// TwinCAT 3 PLC project Untitled1
// ProgramVersion: 3.1.4023.0
// libraries:
//   Tc2_Standard, * (Beckhoff Automation GmbH)
//   Tc2_System, * (Beckhoff Automation GmbH)
//   Tc2_Utilities, * (Beckhoff Automation GmbH)
//   Tc3_Database, * (Beckhoff Automation GmbH)
//   Tc3_EventLogger, * (Beckhoff Automation GmbH)
//   Tc3_Module, * (Beckhoff Automation GmbH)
// project tree:
//   DUTs/DataFlowManagement/ ST_NovRam.TcDUT
//   DUTs/DataFlowManagement/ST_NovRam_SubST/ E_DB_StructureType.TcDUT, ST_NovRam_Status.TcDUT, ST_FileRingBuffer_Status.TcDUT
//   DUTs/ErrHandle/ E_DataBaseTable.TcTLEO
//   DUTs/ E_DataBaseStatus.TcDUT, E_DBID.TcDUT, E_DB_DataType.TcDUT, E_RegularCheckSensorResult.TcDUT, ST_AlarmInfo_DB.TcDUT, ST_AlarmInfo_DB_save.TcDUT, ST_HardwareConfigure_DB.TcDUT, ST_MachineInformation.TcDUT, ST_MachineParameter.TcDUT, ST_MessageElement.TcDUT, ST_OEE_ProductionReport.TcDUT, ST_OEE_ProductionSummary.TcDUT, ST_RegularCheck_Results.TcDUT, ST_RegularCheck_Results_DB.TcDUT, ST_ShopOrderInformation.TcDUT, ST_SoDuration.TcDUT, ST_StopCount.TcDUT
//   DUTs/PHI/ ST_CmdPara_PHI_DB.TcDUT, ST_Inspection_DB.TcDUT, ST_PHI_GroupData_DB.TcDUT, ST_Production_History_DB.TcDUT, ST_Production_History_DB_Test.TcDUT
//   GVLs/ GVL.TcGVL
//   / PlcTask.TcTTO, Task_Consumer.TcTTO
//   POUs/ CheckBounds.TcPOU, MAIN.TcPOU, PG_AddData.TcPOU, PG_SaveData.TcPOU
//   POUs/DataFlow/Lv1/ FB_DataFlowManagement.TcPOU
//   POUs/DataFlow/Lv2/ FB_DataToNovRam.TcPOU, FB_FileRingBufferToDB.TcPOU, FB_NovRamToFileRingBuffer.TcPOU
//   POUs/DataFlow/Lv3%28DB%29/Lv1/ FB_DataUpload_Leo.TcPOU (not stored)
//   POUs/DataFlow/Lv3%28DB%29/Lv2/Background/ FB_CheckDBconnection_DB.TcPOU (not stored)
//   POUs/DataFlow/Lv3%28DB%29/Lv2/DB/ FB_AlarmHistory_DB.TcPOU (not stored), FB_OEE_ProductionReport_DB.TcPOU (not stored), FB_OEE_ProductionSummary_DB.TcPOU (not stored), FB_ProductionHistoryInspection_DB.TcPOU (not stored), FB_Regular_Check_Results_DB.TcPOU (not stored), FB_SoDuration_DB.TcPOU (not stored), FB_StopCount_DB.TcPOU (not stored)
// real-time tasks:
//   TASK PlcTask: cycle T#1ms, priority 20, ADS port 350
//   TASK Task 4: cycle T#1ms, priority 1, ADS port 351

CONFIGURATION Untitled1
    RESOURCE PLC ON TwinCAT3
        TASK PlcTask(INTERVAL := T#1ms, PRIORITY := 20);
        TASK Task_Consumer(INTERVAL := T#1ms, PRIORITY := 1);
        PROGRAM MAIN WITH PlcTask : MAIN;
        PROGRAM PG_AddData WITH PlcTask : PG_AddData;
        PROGRAM PG_SaveData WITH Task_Consumer : PG_SaveData;
    END_RESOURCE
END_CONFIGURATION

// ---- DUTs/DataFlowManagement/ST_NovRam.TcDUT
TYPE ST_NovRam :
STRUCT
	
	//Status
	//NovRam_Status:ST_NovRam_Status;
	arrNovRam_Status:ARRAY[0..6] OF ST_NovRam_Status;
	//FileRingBuffer_Status:ST_FileRingBuffer_Status;
	arrFileRingBuffer_Status:ARRAY[0..6] OF ST_FileRingBuffer_Status;
	
	
	
	//Compressed DATA
	AlarmHistory:ARRAY [0..GVL.NovRamBufferRatio-1] OF ARRAY [0..GVL.arrArrayLength[E_DB_StructureType.AlarmHistory]-1] OF ST_AlarmInfo_DB_save;
	ProductionHistory:ARRAY [0..GVL.NovRamBufferRatio-1] OF ARRAY [0..GVL.arrArrayLength[E_DB_StructureType.ProductionHistory]-1] OF ST_PHI_GroupData_DB;
	ProductionReport:ARRAY [0..GVL.NovRamBufferRatio-1]OF ARRAY [0..GVL.arrArrayLength[E_DB_StructureType.ProductionReport]-1] OF ST_OEE_ProductionReport;
	ProductionSummary:ARRAY [0..GVL.NovRamBufferRatio-1]OF ARRAY [0..GVL.arrArrayLength[E_DB_StructureType.ProductionSummary]-1] OF ST_OEE_ProductionSummary;
	SoDuration:ARRAY [0..GVL.NovRamBufferRatio-1]OF ARRAY [0..GVL.arrArrayLength[E_DB_StructureType.SoDuration]-1] OF ST_SoDuration;
	StopCount:ARRAY [0..GVL.NovRamBufferRatio-1]OF ARRAY [0..GVL.arrArrayLength[E_DB_StructureType.StopCount]-1] OF ST_StopCount;
	RegularCheckResults:ARRAY [0..GVL.NovRamBufferRatio-1]OF ARRAY [0..GVL.arrArrayLength[E_DB_StructureType.RegularCheckResults]-1] OF ST_RegularCheck_Results;
	

END_STRUCT
END_TYPE

// ---- DUTs/DataFlowManagement/ST_NovRam_SubST/E_DB_StructureType.TcDUT
{attribute 'qualified_only'}
{attribute 'strict'}
TYPE E_DB_StructureType :
(
	AlarmHistory := 0,
	ProductionHistory := 1,
	ProductionReport := 2,
	ProductionSummary := 3,
	SoDuration:=4,
	StopCount:=5,
	RegularCheckResults:=6
);
END_TYPE

// ---- DUTs/DataFlowManagement/ST_NovRam_SubST/ST_NovRam_Status.TcDUT
TYPE ST_NovRam_Status :
STRUCT
	nowRowIndex:UDINT;
	writenIndex:UDINT;
	RowDataLocked:ARRAY[0..GVL.NovRamBufferRatio-1]OF BOOL;
	writenCount:UDINT;//1217
	
END_STRUCT
END_TYPE

// ---- DUTs/DataFlowManagement/ST_NovRam_SubST/ST_FileRingBuffer_Status.TcDUT
TYPE ST_FileRingBuffer_Status :
STRUCT
	bFileFull:ARRAY[0..GVL.NovRamBufferRatio-1] OF ARRAY [0..GVL.FileRingBufferRatio-1] OF BOOL;//9
	
	//FileRingBufferLocked:ARRAY[0..GVL.FileRingBufferTotalNum-1]OF BOOL;
	nowFileIndex:ARRAY [0..gvl.FileRingBufferRatio-1] OF UDINT;//3
END_STRUCT
END_TYPE

// ---- DUTs/ErrHandle/E_DataBaseTable.TcTLEO
{attribute 'qualified_only'}
{attribute 'to_string'}
TYPE E_DataBaseTable :
(
	NoError := 0,
	HardwareConfig_ReadFail,
	HardwareConfig_ReadDataOutOfRange,
	HardwareConfig_InputReferenceInvaild,
	HardwareConfig_NoData,
	MachineParameter_ReadFail,
	MachineParameter_ReadDataOutOfRange,
	MachineParameter_InputReferenceInvaild,
	MachineParameter_NoData,
	MachineParameter_FillDataToSubsysFail,
	MachineParameter_FillDataToCoreSysFail,
	MachineParameter_FillDataToMachineFail,
	MessageList_ReadFail,
	MessageList_ReadDataOutOfRange,	
	MessageList_InputReferenceInvaild,
	MessageList_NoData,
	MessageList_MessageCodeOrArraySizeOutOfRange,
	AlarmHistory_UploadDataFail,
	DataUpload_ConnectToDBFail,
	DataUpload_AlarmHistoryBufferFull,
	DataUpload_AlarmHistoryUploadFail,
	DataUpload_AlarmHistoryUploadFailWriteDataToFileFail, //重大異常，不能直接reset需要人員排查原因，程式內部鎖死不能reset
	DataUpload_ProductionHistoryBufferFull,
	DataUpload_ProductionHistoryUploadFail,
	DataUpload_ProductionHistoryWriteDataToFileFail, //重大異常，不能直接reset需要人員排查原因，程式內部鎖死不能reset
	DataUpload_ProductionReportBufferFull,
	DataUpload_ProductionReportUploadFail,
	DataUpload_ProductionReportWriteDataToFileFail, //重大異常，不能直接reset需要人員排查原因，程式內部鎖死不能reset
	DataUpload_ProductionSummaryBufferFull,
	DataUpload_ProductionSummaryUploadFail,
	DataUpload_ProductionSummaryWriteDataToFileFail, //重大異常，不能直接reset需要人員排查原因，程式內部鎖死不能reset
	DataUpload_SoDurationBufferFull,
	DataUpload_SoDurationUploadFail,
	DataUpload_SoDurationWriteDataToFileFail, //重大異常，不能直接reset需要人員排查原因，程式內部鎖死不能reset
	DataUpload_StopCountBufferFull,	
	DataUpload_StopCountUploadFail,
	DataUpload_StopCountWriteDataToFileFail, //重大異常，不能直接reset需要人員排查原因，程式內部鎖死不能reset
	DataUpload_RegularCheckResultsBufferFull,
	DataUpload_RegularCheckResultsUploadFail,
	DataUpload_RegularCheckResultsWriteDataToFileFail, //重大異常，不能直接reset需要人員排查原因，程式內部鎖死不能reset
	ProductionReport_UploadDataFail,
	ProductionSummary_UploadDataFail,
	ProductionHistoryInspection_UploadDataFail,
	RegularCheckResults_UploadDataFail,
	SoDuration_UploadDataFail,
	StopCount_UploadDataFail,
	CheckDBconnection_ReadDBStatusTimeout,
	CheckDBconnection_RetryConnectToDBFail,
	CheckDBconnection_StatusDataOutOfRange,
	ProdHistoryProcedure_UploadDataFail,
	ProdHistoryProcedure_WriteDataToFileFail, //重大異常，不能直接reset需要人員排查原因，程式內部鎖死不能reset
	ProdHistoryProcedure_InputInterfaceInvalid,
	ProdStatusChangedStopCount_FillDataTimeout,
	ProdStatusChangedStopCount_AddDataToBufferTimeout,
	UploadEndBatchData_FillProductionReportDataTimeout,
	UploadEndBatchData_FillProductionSummaryDataTimeout,
	UploadEndBatchData_FillSoDurationDataTimeout,
	UploadEndBatchData_AddProductionReportDataToBufferTimeout,
	UploadEndBatchData_AddProductionSummaryDataToBufferTimeout,
	UploadEndBatchData_AddSoDurationDataToBufferTimeout,
	UploadProdRegularReport_FillProductionReportDataTimeout,
	UploadProdRegularReport_AddProductionReportDataToBufferTimeout
	
	
)UDINT;
END_TYPE

// ---- DUTs/E_DataBaseStatus.TcDUT
{attribute 'qualified_only'}
{attribute 'to_string'}
TYPE E_DataBaseStatus :
(
	ONLINE := 0,
	RESTORING,
	RECOVERING,
	RECOVERY_PENDING,
	SUSPECT,
	EMERGENCY,
	OFFLINE,
	COPYING,
	OFFLINE_SECONDARY
)USINT;
END_TYPE

// ---- DUTs/E_DBID.TcDUT
{attribute 'qualified_only'}
{attribute 'to_string'}
TYPE E_DBID :
(
	BypassDB	:= 0,
	RemoteDB  	:= 1,
	LocalDB		:= 2
)UDINT;
END_TYPE

// ---- DUTs/E_DB_DataType.TcDUT
{attribute 'qualified_only'}
{attribute 'to_string'}
TYPE E_DB_DataType :
(
	Double := 0,
	StringType,
	Ring,
	Boolean,
	I32,
	U32,
	DynamicRing
)INT;
END_TYPE

// ---- DUTs/E_RegularCheckSensorResult.TcDUT
{attribute 'qualified_only'}
{attribute 'to_string'}
TYPE E_RegularCheckSensorResult :
(
	Null, // 感測器沒判定過/使用  DB寫Null
	Pass, // 判定結果為OK  DB寫1
	Fail // 判定結果為NG  DB寫0
);
END_TYPE

// ---- DUTs/PHI/ST_CmdPara_PHI_DB.TcDUT
TYPE ST_CmdPara_PHI_DB :
	STRUCT
		//Product History
		dt_start_time            : DT ;
		r_duration               : REAL ;
		dt_end_time              : DT ;
		di_station_number        : DINT ;
		wstr_station_name        : WSTRING(255) ; //20221107
		di_track_number          : DINT ;
		di_wpc_number            : DINT ;
		b_part_ok_overal_results : BOOL ;
		str_so_number            : STRING(12) ;
		str_faam_id              : STRING(20) ;
		di_so_id                 : DINT ;
		
		//1st Inspection
		di_sub_station_number_1 : DINT ;
		str_sensor_type_1       : STRING(50) ;
		b_inspection_results_1  : BOOL ;
		r_inspection_value_1    : REAL ;
		str_faam_id_1           : STRING(20) ;
		str_so_number_1         : STRING(12) ;
		
		//2nd Inspection
		di_sub_station_number_2 : DINT ;
		str_sensor_type_2       : STRING(50) ;
		b_inspection_results_2  : BOOL ;
		r_inspection_value_2    : REAL ;
		str_faam_id_2           : STRING(20) ;
		str_so_number_2         : STRING(12) ;
		
		//3nd Inspection
		di_sub_station_number_3 : DINT ;
		str_sensor_type_3       : STRING(50) ;
		b_inspection_results_3  : BOOL ;
		r_inspection_value_3    : REAL ;
		str_faam_id_3           : STRING(20) ;
		str_so_number_3         : STRING(12) ;
		
		//4nd Inspection
		di_sub_station_number_4 : DINT ;
		str_sensor_type_4	     : STRING(50) ;
		b_inspection_results_4  : BOOL ;
		r_inspection_value_4    : REAL ;
		str_faam_id_4           : STRING(20) ;
		str_so_number_4         : STRING(12) ;
		
		//5nd Inspection
		di_sub_station_number_5 : DINT ;
		str_sensor_type_5       : STRING(50) ;
		b_inspection_results_5  : BOOL ;
		r_inspection_value_5    : REAL ;
		str_faam_id_5           : STRING(20) ;
		str_so_number_5         : STRING(12) ;
	END_STRUCT
END_TYPE

// ---- DUTs/PHI/ST_Inspection_DB.TcDUT
TYPE ST_Inspection_DB : // Sensor inspection information and result
	STRUCT
		diSub_station_number 	: DINT ;			// 站點上第N組感測器
		sSensor_type        	: STRING(50) ;	// Sensor類型
		bInspection_results 	: BOOL ;			// Sensor回傳結果
		rInspection_value   	: REAL ;			// Sensor回傳數值
		sFaam_id            	: STRING(20) ;
		sSo_number          	: STRING(12) ;
		//product_history_id 	: LINT ;
	END_STRUCT
END_TYPE

// ---- DUTs/PHI/ST_PHI_GroupData_DB.TcDUT
 //Product History and Inspection data
 //X64 size: 1064 bytes
TYPE ST_PHI_GroupData_DB : //Production information of the station, including single production data and sensor results
	STRUCT
		stProductHistory        						: ST_Production_History_DB ; // single production data
		arrstInspection         						: ARRAY[1..5] OF ST_Inspection_DB ; //max sensor number = 5
		arrbInspectionResultHaveSensorValue           	: ARRAY[1..5] OF BOOL ; // return data of the sensor have a numerical value
	END_STRUCT
END_TYPE

// ---- DUTs/PHI/ST_Production_History_DB.TcDUT
TYPE ST_Production_History_DB : // single production data of a station
	STRUCT
		dtStart_time             	: DT ;					// 作業開始時間
		rDuration               	: REAL ;				// unit: sec    (end_time - start_time)
		dtEnd_time               	: DT ;					// 作業結束時間
		diStation_number         	: DINT ;				// 站點編號
		wsStation_name           	: WSTRING(255) ; 		// 站點名稱
		diTrack_number           	: DINT ;				// 未定義  Smart Hardcode為1
		diWpc_number            	: DINT ;				// Shuttle Id
		bPart_ok_overal_results 	: BOOL ;				// 此站點最終判斷/作業結果為OK或NG (彙整站點上的感測器結果及作業結果)
		sSo_number              	: STRING(12) ;			// 由HMI透過ADS告知  (DB中的So資料表需要存在對應資料)
		sFaam_id                	: STRING(20) ;			// 由DB讀取
		diSo_id                  	: DINT ;				// 由HMI透過ADS告知 (DB中的So資料表需要存在對應資料)
	END_STRUCT
END_TYPE

// ---- DUTs/PHI/ST_Production_History_DB_Test.TcDUT
TYPE ST_Production_History_DB_Test: // single production data of a station
	STRUCT
		dtStart_time             	: DT ;					// 作業開始時間
		rDuration               	: REAL ;				// unit: sec    (end_time - start_time)
		dtEnd_time               	: DT ;					// 作業結束時間
		usiStation_number         	: USINT ;				// 站點編號
		sStation_name           	: STRING(50) ; 		// 站點名稱
		usiTrack_number           	: USINT ;				// 未定義  Smart Hardcode為1
		usiWpc_number            	: USINT ;				// Shuttle Id
		bPart_ok_overal_results 	: BOOL ;				// 此站點最終判斷/作業結果為OK或NG (彙整站點上的感測器結果及作業結果)
		sSo_number              	: STRING(12) ;			// 由HMI透過ADS告知  (DB中的So資料表需要存在對應資料)
		sFaam_id                	: STRING(20) ;			// 由DB讀取
		diSo_id                  	: DINT ;				// 由HMI透過ADS告知 (DB中的So資料表需要存在對應資料)
	END_STRUCT
END_TYPE

// ---- DUTs/ST_AlarmInfo_DB.TcDUT
// X64 size: 4984 byte
TYPE ST_AlarmInfo_DB :
STRUCT
	lrTime_ms    	: LREAL ;		
	iMsgProc    	: INT ;			// 未明 先填1
	iStateAfter 	: INT ;			// 1: Error trigger  0: reset
	iMsgClass   	: INT ;			// 1: error 2: warning 3: msg
	diMsgNumber  	: DINT ;		// MsgCode等同於ErrorId
	wsVar1			: WSTRING(255);	// 備註1(可不填)
	wsVar2			: WSTRING(255);	// 備註2(可不填)
	wsVar3			: WSTRING(255);	// 備註3(可不填)
	wsVar4			: WSTRING(255);	// 備註4(可不填)
	wsVar5			: WSTRING(255);	// 備註5(可不填)
	wsVar6			: WSTRING(255);	// 備註6(可不填)
	wsVar7			: WSTRING(255);	// 備註7(可不填)
	wsVar8			: WSTRING(255);	// 備註8(可不填)
	sTimeString 	: STRING(25); 	// Data Format: '2023-08-15 15:11:14'  		// SQL Database為char type 26bytes 
	wsMsgText    	: WSTRING(255); // 文字訊息(顯示在HMI給使用者看的訊息)
	sPLC        	: STRING(255); 	// Data Format: 'CoreSys' 
	wsEquipment  	: WSTRING(25);
	sFaam_id    	: STRING(20);
	
END_STRUCT
END_TYPE

// ---- DUTs/ST_AlarmInfo_DB_save.TcDUT
// X64 size: 680 byte
TYPE ST_AlarmInfo_DB_save:
STRUCT
	(*
	lrTime_ms    	: LREAL ;		
	siMsgProc    	: SINT ;			// 未明 先填1
	siStateAfter 	: SINT ;			// 1: Error trigger  0: reset
	siMsgClass   	: SINT ;			// 1: error 2: warning 3: msg
	diMsgNumber  	: DINT ;		// MsgCode等同於ErrorId
	//wsVar1			: WSTRING(255);	// 備註1(可不填)
	//wsVar2			: WSTRING(255);	// 備註2(可不填)
	//wsVar3			: WSTRING(255);	// 備註3(可不填)
	//wsVar4			: WSTRING(255);	// 備註4(可不填)
	//wsVar5			: WSTRING(255);	// 備註5(可不填)
	//wsVar6			: WSTRING(255);	// 備註6(可不填)
	//wsVar7			: WSTRING(255);	// 備註7(可不填)
	//wsVar8			: WSTRING(255);	// 備註8(可不填)
	sTimeString 	: STRING(25); 	// Data Format: '2023-08-15 15:11:14'  		// SQL Database為char type 26bytes 
	wsMsgText    	: WSTRING(255); // 文字訊息(顯示在HMI給使用者看的訊息)
	sPLC        	: STRING(50); 	// Data Format: 'CoreSys' 
	wsEquipment  	: WSTRING(25);
	sFaam_id    	: STRING(20);
	*)
	lrTime_ms    	: LREAL ;		
	iMsgProc    	: INT ;			// 未明 先填1
	iStateAfter 	: INT ;			// 1: Error trigger  0: reset
	iMsgClass   	: INT ;			// 1: error 2: warning 3: msg
	diMsgNumber  	: DINT ;		// MsgCode等同於ErrorId
	sTimeString 	: STRING(25); 	// Data Format: '2023-08-15 15:11:14'  		// SQL Database為char type 26bytes 
	wsMsgText    	: WSTRING(255); // 文字訊息(顯示在HMI給使用者看的訊息)
	sPLC        	: STRING(255); 	// Data Format: 'CoreSys' 
	wsEquipment  	: WSTRING(25);
	sFaam_id    	: STRING(20);
END_STRUCT
END_TYPE

// ---- DUTs/ST_HardwareConfigure_DB.TcDUT
TYPE ST_HardwareConfigure_DB :
STRUCT
	iParametersID			: INT;
	wsConfigureItem			: WSTRING(255);
	wsConfigureName			: WSTRING(255);
	wsConfigureValue		: WSTRING(255);
	wsDataType				: WSTRING(255);
	wsDescription			: WSTRING(255);
END_STRUCT
END_TYPE

// ---- DUTs/ST_MachineInformation.TcDUT
TYPE ST_MachineInformation :
STRUCT
	sFaam_id                  : STRING(20) ;	// 設備ID
	wsEquipment               : WSTRING(25) ;	// 設備名稱
END_STRUCT
END_TYPE

// ---- DUTs/ST_MachineParameter.TcDUT
// Generated by SQL Query Editor
TYPE ST_MachineParameter :
STRUCT
	iParameters_Index	: INT;
	wsTag_Name			: WSTRING(255);
	iStation			: INT;
	wsParameters_Unit	: WSTRING(50);
	iPackTagID			: INT;
	wsParameters_Value	: WSTRING(255);
	eDataType			: E_DB_DataType;
END_STRUCT
END_TYPE


//SQL Command
(*
SELECT          Global_Machine_Parameters.Parameters_Index, 
				Global_Machine_Parameters.Parameters_Name, 
				Global_Machine_Parameters.Station, 
				Global_Machine_Parameters.Parameters_Unit,
                Global_Machine_Parameters.PackTagID, 
				Global_Machine_Parameters_Value.Parameters_Value
FROM            Global_Machine_Parameters_Value INNER JOIN
                Global_Machine_Parameters ON 
                Global_Machine_Parameters_Value.Parameters_Index = Global_Machine_Parameters.Parameters_Index
ORDER BY Global_Machine_Parameters.Parameters_Index
*)

// ---- DUTs/ST_MessageElement.TcDUT
// X64 Size: 2052 byte
TYPE ST_MessageElement :
STRUCT
	iCode						: INT;			// MsgCode (ErrorCode)
	wsCategory					: WSTRING(255); // 文字訊息分類 EX: "Safety Message", "Beaker and Bin and Drawer Message" etc.
	wsItem						: WSTRING(255);	// 此訊息的項目名稱，通常會與wsFirst_Language_Message重複
	wsFirst_Language_Message  	: WSTRING(255); // 多國語言1文字訊息(此項為預設值 內文為英文)
	wsSecond_Language_Message 	: WSTRING(255); // 多國語言2文字訊息(內文為中文或其他)
	iMessage_Type 				: INT;
END_STRUCT
END_TYPE

// ---- DUTs/ST_OEE_ProductionReport.TcDUT
// X64 size: 172 bytes
TYPE ST_OEE_ProductionReport :
	STRUCT
		wsOee_equipment            	: WSTRING(25) ;
		dtTime_start               	: DT ;
		dtTime_end                 	: DT ;
		diAverage_ppm              	: DINT ;
		diIdeal_production         	: DINT ;
		diOk_part_count            	: DINT ;
		rTotal_idle_time          	: REAL ;
		diReal_production          	: DINT ;
		diGood_parts               	: DINT ;
		rGood_parts_percentage    	: REAL ;
		diQuantity_loss            	: DINT ;
		rQuantity_loss_percentage 	: REAL ;
		rPm                       	: REAL ;
		rYm                       	: REAL ;
		rAm                       	: REAL ;
		rEm                       	: REAL ;
		rOm                       	: REAL ;
		rAvailable_time           	: REAL ;
		rSchedule_loss            	: REAL ;
		rRunning_time             	: REAL ;
		rDowntime_loss            	: REAL ;
		sFaam_id                  	: STRING(20) ;
		sSo_number               	: STRING(12) ;
		diSo_id                    	: DINT ;
	END_STRUCT
END_TYPE

// ---- DUTs/ST_OEE_ProductionSummary.TcDUT
// X64 size: 148 bytes
TYPE ST_OEE_ProductionSummary :
	STRUCT
		wsEquipment     : WSTRING(20) ;
		wsSummary_type  : WSTRING(30) ;
		diSummary_value : DINT ;
		sFaam_id       : STRING(20) ;
		sSo_number     : STRING(12) ;
		diSo_id         : DINT ;
	END_STRUCT
END_TYPE

// ---- DUTs/ST_RegularCheck_Results.TcDUT
// X64 size: 572 bytes
TYPE ST_RegularCheck_Results :
	STRUCT
		diStation_number          	: DINT ;
		diTrack_number            	: DINT ;
		dtStart_time              	: DT ;
		eSensor                  	: E_RegularCheckSensorResult ;
		eCamera                  	: E_RegularCheckSensorResult ;
		eLoadcell                	: E_RegularCheckSensorResult ;
		eSensor2                 	: E_RegularCheckSensorResult ;
		diRegular_check_id        	: DINT ;
		sFaam_id                 	: STRING(20) ;
		sSo_number               	: STRING(12) ;
		diSo_id                   	: DINT ;
		wsEmployee_name_logged_in 	: WSTRING(255) ;
	END_STRUCT
END_TYPE

// ---- DUTs/ST_RegularCheck_Results_DB.TcDUT
// X64 size: 572 bytes
TYPE ST_RegularCheck_Results_DB :
	STRUCT
		diStation_number          	: DINT ;
		diTrack_number            	: DINT ;
		dtStart_time              	: DT ;
		bSensor                  	: BOOL ;
		bCamera                  	: BOOL ;
		bLoadcell                	: BOOL ;
		bSensor2                 	: BOOL ;
		diRegular_check_id        	: DINT ;
		sFaam_id                 	: STRING(20) ;
		sSo_number               	: STRING(12) ;
		diSo_id                   	: DINT ;
		wsEmployee_name_logged_in 	: WSTRING(255) ;
	END_STRUCT
END_TYPE

// ---- DUTs/ST_ShopOrderInformation.TcDUT
TYPE ST_ShopOrderInformation :
STRUCT
	diSo_id                    	: DINT ;
	sSo_number               	: STRING(12) ;
END_STRUCT
END_TYPE

// ---- DUTs/ST_SoDuration.TcDUT
// X64 size: 2100 bytes
TYPE ST_SoDuration :
	STRUCT
		dtBatch_start_time            	: DT ;
		dtBatch_end_time              	: DT ;
		//bNormal_complition           	: BOOL ; //改放至最後才寫  放在這位置寫入DB時會導致下個資料WString在DB裡開頭多一個空白byte的資料
		wsBatch_end_reason             	: WSTRING(255) ;
		wsBatch_end_reason_description 	: WSTRING(255) ;
		wsEmployee_name_start_user     	: WSTRING(255) ;
		wsEmployee_name_end_user       	: WSTRING(255) ;
		sSo_number                    	: STRING(12) ;
		sFaam_id                      	: STRING(20) ;
		diSo_id                        	: DINT ;
		bNormal_complition           	: BOOL ;
	END_STRUCT
END_TYPE

// ---- DUTs/ST_StopCount.TcDUT
TYPE ST_StopCount :
	STRUCT
		dtStart_time              : DT ;
		dtEnd_time                : DT ;
		wsEmployee_name_logged_in : WSTRING(255) ;
		sStop_reason             : STRING(3) ;
		sAssembly_income_code    : STRING(16) ;
		sSo_number               : STRING(12) ;
		sFaam_id                 : STRING(20) ;
		diSo_id                   : DINT ;
		wsEquipment               : WSTRING(25) ;
	END_STRUCT
END_TYPE

// ---- GVLs/GVL.TcGVL
{attribute 'qualified_only'}
VAR_GLOBAL CONSTANT//NovRam Management
		
	Max_IndexNum:UDINT:=40;//Index數量

	//File大小
	//fileRingBufferSize:UDINT:=50*1000;//Byte
	arrFileRingBufferSize:ARRAY [0..6] OF UDINT:=[
	100*1000,//Alarm History
	100*1000,//Production History
	100*1000,//ProductionReport
	100*1000,//ProductionSummary
	100*1000,//SoDuration
	100*1000,//StopCount
	100*1000//RegularCheckResults
	];
	
	//資料的陣列長度
	//AlarmHistory_ArrayLength:UDINT:=30;
	//ProductionHistory_ArrayLength:UDINT:=30;
	arrArrayLength:ARRAY[0..6] OF UDINT:=[
	30,//Alarm History
	30,//Production History
	30,//ProductionReport
	30,//ProductionSummary
	30,//SoDuration
	30,//StopCount
	30//RegularCheckResults
	];
	
	//NovRam中Array數量
	NovRamBufferRatio:UDINT:=3;
	//arrNovRamBufferRatio:ARRAY [0..1] OF UDINT:=[
	//3,//Alarm History
	//3//Production History
	//];
	
	//單一NovRam Array對應的File數量
	FileRingBufferRatio:UDINT:=3;
	//arrFileRingBufferRatio:ARRAY[0..1] OF UDINT:=[
	//10,//Alarm History
	//10//Production History
	//];
	
	//fileFolder:STRING(255):='c:\_Yenlin\';
	arrFileFolder:ARRAY [0..6] OF STRING(255):=[
	'c:\_Yenlin\',//Alarm History
	'c:\_Yenlin\',//Production History
	'c:\_Yenlin\',//ProductionReport
	'c:\_Yenlin\',//ProductionSummary
	'c:\_Yenlin\',//SoDuration
	'c:\_Yenlin\',//StopCount
	'c:\_Yenlin\'//RegularCheckResults
	];
	
	
END_VAR

VAR_GLOBAL
	fbDataFlowManagement:FB_DataFlowManagement;
	udiUpperCnt : UDINT;
	udiLowerCnt	: UDINT;
END_VAR

// ---- POUs/MAIN.TcPOU
PROGRAM MAIN
VAR
	i:UDINT;
	
END_VAR

END_PROGRAM

// ---- POUs/PG_AddData.TcPOU
PROGRAM PG_AddData
VAR
	i:UDINT;
	repeatTimer:TON;
	
	
	AlarmHistoryData_Write:ST_AlarmInfo_DB;
	ProductionHistoryData_Write:ST_PHI_GroupData_DB;
	ProductionReport_Write:ST_OEE_ProductionReport;
	ProductionSummary_Write:ST_OEE_ProductionSummary;
	SoDuration_Write:ST_SoDuration;
	StopCount_Write:ST_StopCount;
	RegularCheckResults_Write:ST_RegularCheck_Results;
	
	
	writeFailCount:UDINT;
	writeFailCount2:UDINT;
	writeFailCount3:UDINT;
	writeFailCount4:UDINT;
	writeFailCount5:UDINT;
	writeFailCount6:UDINT;
	writeFailCount7:UDINT;
	
	//
	bDoWrite:BOOL;
	k:UDINT;
	udiWriteCount:UDINT;
END_VAR


//simulate that Peak Data amount as 500 ms
repeatTimer(IN:=TRUE,PT:=T#300MS);

IF repeatTimer.Q THEN
	
	repeatTimer(in:=FALSE);
	
		
	FOR i:=1 TO 10 DO
		
		IF bDoWrite THEN
			//bDoWrite:=FALSE;
			//(*
				AlarmHistoryData_Write.wsMsgText:="20231217_2130";
				IF GVL.fbDataFlowManagement.M_Add_AlarmHistory(addData:=AlarmHistoryData_Write) = FALSE THEN
					writeFailCount:=writeFailCount+1;
				END_IF
				udiWriteCount:=udiWriteCount+1;
			//*)
		END_IF
		
		
		(*
		
		ProductionHistoryData_Write.stProductHistory.sSo_number:= 'Fred';				// From ADS  //需要對應DB的So表的So_Number
		ProductionHistoryData_Write.stProductHistory.sFaam_id:= 'FB000120-E002-0001';		// from DB
		ProductionHistoryData_Write.stProductHistory.diSo_id:= 3736;			// from ADS  //需要對應DB的So表So_id
		ProductionHistoryData_Write.stProductHistory.diTrack_number:= 998877;
		IF GVL.fbDataFlowManagement.M_Add_ProductionHistoryInspection(addData:=ProductionHistoryData_Write) = FALSE THEN
			writeFailCount2:=writeFailCount2+1;
		END_IF
		*)
		(*
		ProductionSummary_Write.diSo_id:=3736;
		ProductionSummary_Write.diSummary_value:=87887;
		IF GVL.fbDataFlowManagement.M_Add_ProductionSummary(addData:=ProductionSummary_Write) = FALSE THEN
			writeFailCount4:=writeFailCount4+1;
		END_IF
		*)
		
		(*
		SoDuration_Write.diSo_id:=3736;
		SoDuration_Write.wsBatch_end_reason:="for test87887";
		IF GVL.fbDataFlowManagement.M_Add_SoDuration(addData:=SoDuration_Write) = FALSE THEN
			writeFailCount5:=writeFailCount5+1;
		END_IF
		*)
		
		(*
		StopCount_Write.diSo_id:=3736;
		StopCount_Write.sStop_reason:='oeL';
		IF GVL.fbDataFlowManagement.M_Add_StopCount(addData:=StopCount_Write) = FALSE THEN
			writeFailCount6:=writeFailCount6+1;
		END_IF
		*)
		
		(*
		ProductionReport_Write.diOk_part_count:=9987;
		ProductionReport_Write.diSo_id:=3736;
		ProductionReport_Write.sSo_number:='Fred';
		ProductionReport_Write.sFaam_id:='FB000120-E002-0001';
		
		IF GVL.fbDataFlowManagement.M_Add_ProductionReport(addData:=ProductionReport_Write) = FALSE THEN
			writeFailCount3:=writeFailCount3+1;
		END_IF
		*)
				
		(*
		RegularCheckResults_Write.diRegular_check_id:=3731;
		RegularCheckResults_Write.diSo_id:=3736;
		RegularCheckResults_Write.wsEmployee_name_logged_in:="Leo8787";
		RegularCheckResults_Write.sSo_number:='Fred';
		RegularCheckResults_Write.sFaam_id:='FB000120-E002-0001';
		IF GVL.fbDataFlowManagement.M_Add_RegularCheckResults(addData:=RegularCheckResults_Write) = FALSE THEN
			writeFailCount7:=writeFailCount7+1;
		END_IF
		*)
	END_FOR
END_IF

END_PROGRAM

// ---- POUs/PG_SaveData.TcPOU
PROGRAM PG_SaveData
VAR
	i:UDINT;
	k:UDINT;
	
	wsDBname				: WSTRING(128) := "Smart"; // 暫時測試用
	eDBID					: E_DBID		:= E_DBID.RemoteDB;
	stSoInfo	: ST_ShopOrderInformation;
	stMachineInfo : ST_MachineInformation;

END_VAR

(*
stSoInfo.diSo_id := stShopOrder_pre.diShopOrderID;
stSoInfo.sSo_number := stShopOrder_pre.sShopOrderNumber;

stMachineInfo.sFaam_id := sEqipmentNumber;
stMachineInfo.wsEquipment := wsEquipment;
*)
GVL.fbDataFlowManagement(eDBID := eDBID,
					wsDBname := wsDBname,
					stMachineInfo := stMachineInfo,
					stSoInfo := stSoInfo,);

END_PROGRAM

// ---- POUs/DataFlow/Lv1/FB_DataFlowManagement.TcPOU
FUNCTION_BLOCK FB_DataFlowManagement
VAR CONSTANT
END_VAR
//NovRam
VAR RETAIN
	NovRamData:ST_NovRam;
END_VAR
VAR_INPUT
	eDBID		: E_DBID := E_DBID.RemoteDB;
	wsDBname	: WSTRING(128); // DB Name
	stMachineInfo : ST_MachineInformation;
	stSoInfo	: ST_ShopOrderInformation;
END_VAR
VAR_OUTPUT
END_VAR
VAR
	//{attribute 'hide'}
	lrFileUseRate: ARRAY[0..6] OF LREAL;
	//{attribute 'hide'}
	lrRamUseRate:ARRAY[0..6] OF LREAL;
	
	//Data To NovRam
	//{attribute 'hide'}
	fbDataToNovRam : FB_DataToNovRam;
	//NovRam To FileRingBuffer
	//{attribute 'hide'}
	fbNovRamToFileRingBuffer:ARRAY [0..6] OF ARRAY[0..GVL.NovRamBufferRatio-1] OF FB_NovRamToFileRingBuffer;
	//FileRingBuffer To DataBase
	//{attribute 'hide'}
	fbFileRingBufferToDB:ARRAY [0..6] OF ARRAY [0..GVL.NovRamBufferRatio-1] OF ARRAY[0..GVL.FileRingBufferRatio-1] OF FB_FileRingBufferToDB;
END_VAR

//FB cyclic
M_CyclicUpdate();

//Calc Use Rate
M_CalcUseRate(lrFileUseRate:=lrFileUseRate,lrRamUseRate:=lrRamUseRate);

METHOD M_Add_AlarmHistory : BOOL
VAR_INPUT
	addData : ST_AlarmInfo_DB ;
END_VAR
M_Add_AlarmHistory:=fbDataToNovRam.M_AlarmHistory(addData:=addData);
END_METHOD

METHOD M_Add_ProductionHistoryInspection : BOOL
VAR_INPUT
	addData:ST_PHI_GroupData_DB;
END_VAR
M_Add_ProductionHistoryInspection:=fbDataToNovRam.M_ProductionHistory(addData:=addData);
END_METHOD

METHOD M_Add_ProductionReport : BOOL
VAR_INPUT
	addData:ST_OEE_ProductionReport;
END_VAR
M_Add_ProductionReport:=fbDataToNovRam.M_ProductionReport(addData:=addData);
END_METHOD

METHOD M_Add_ProductionSummary : BOOL
VAR_INPUT
	addData:ST_OEE_ProductionSummary;
END_VAR
M_Add_ProductionSummary:=fbDataToNovRam.M_ProductionSummary(addData:=addData);
END_METHOD

METHOD M_Add_RegularCheckResults : BOOL
VAR_INPUT
	addData:ST_RegularCheck_Results;
END_VAR
M_Add_RegularCheckResults:=fbDataToNovRam.M_RegularCheckResults(addData:=addData);
END_METHOD

METHOD M_Add_SoDuration : BOOL
VAR_INPUT
	addData:ST_SoDuration;
END_VAR
M_Add_SoDuration:=fbDataToNovRam.M_SoDuration(addData:=addData);
END_METHOD

METHOD M_Add_StopCount : BOOL
VAR_INPUT
	addData:ST_StopCount;
END_VAR
M_Add_StopCount:=fbDataToNovRam.M_StopCount(addData:=addData);
END_METHOD

METHOD M_AutoFill_MachineInfo : BOOL
VAR_INPUT
	refsFaam_id		: REFERENCE TO STRING(20); // 設備ID
	refwsEquipment : REFERENCE TO WSTRING(25); // 設備名稱
END_VAR
(*
IF __ISVALIDREF(refwsEquipment) AND_THEN refwsEquipment = "" THEN //檢查Equipmet是否有填值
	refwsEquipment := stMachineInfo.wsEquipment;
END_IF

IF __ISVALIDREF(refsFaam_id) AND_THEN refsFaam_id = '' THEN //檢查Equipmet是否有填值
	refsFaam_id := stMachineInfo.sFaam_id;
END_IF

M_AutoFill_MachineInfo := True;
*)
END_METHOD

METHOD M_AutoFill_SoInfo : BOOL
VAR_INPUT
	refdiSo_id	: REFERENCE TO DINT;
	refsSo_number : REFERENCE TO STRING(12);
END_VAR
(*
IF __ISVALIDREF(refdiSo_id) AND_THEN refdiSo_id = 0 THEN
	refdiSo_id := stSoInfo.diSo_id;
END_IF

IF __ISVALIDREF(refsSo_number) AND_THEN refsSo_number = '' THEN
	refsSo_number := stSoInfo.sSo_number;
END_IF

M_AutoFill_SoInfo := True;
*)
END_METHOD

METHOD PRIVATE M_CalcUseRate : BOOL
VAR_IN_OUT
	lrFileUseRate: ARRAY[0..6] OF LREAL;
	lrRamUseRate:ARRAY[0..6] OF LREAL;
END_VAR
VAR
	iStruType:UDINT;
	iRamIndex:UDINT;iFileIndex:UDINT;
	
	udiRamFullCount:UDINT;
	udiFileFullCount:UDINT;
END_VAR
FOR iStruType:=0 TO 6 DO
	
	udiRamFullCount:=0;
	udiFileFullCount:=0;
	
	FOR iRamIndex:=0 TO GVL.NovRamBufferRatio-1 DO
		
		IF NovRamData.arrNovRam_Status[iStruType].RowDataLocked[iRamIndex] THEN//ram
			udiRamFullCount:=udiRamFullCount+1;
		END_IF
		
		FOR iFileIndex:=0 TO GVL.FileRingBufferRatio-1 DO//file
			IF NovRamData.arrFileRingBuffer_Status[iStruType].bFileFull[iRamIndex][iFileIndex] = TRUE THEN
				udiFileFullCount:=udiFileFullCount+1;
			END_IF
		END_FOR
	END_FOR
	
	lrFileUseRate[iStruType]:=UDINT_TO_LREAL(udiFileFullCount) 
								/ (UDINT_TO_LREAL(GVL.NovRamBufferRatio) * UDINT_TO_LREAL(GVL.FileRingBufferRatio));
	lrRamUseRate[iStruType]:=UDINT_TO_LREAL(udiRamFullCount) / UDINT_TO_LREAL(GVL.NovRamBufferRatio);
END_FOR
END_METHOD

METHOD PRIVATE M_CyclicUpdate : BOOL
VAR_INPUT
END_VAR
VAR
	i:UDINT;k:UDINT;
END_VAR
//Data to NovRam
fbDataToNovRam(NovRamData:=NovRamData);


//NovRam to File
FOR i:= 0 TO GVL.NovRamBufferRatio-1 DO
	fbNovRamToFileRingBuffer[E_DB_StructureType.AlarmHistory][i](udiNovRamIndex:=i,dataType:=E_DB_StructureType.AlarmHistory,NovRamData:=NovRamData);
	fbNovRamToFileRingBuffer[E_DB_StructureType.ProductionHistory][i](udiNovRamIndex:=i,dataType:=E_DB_StructureType.ProductionHistory,NovRamData:=NovRamData);
	fbNovRamToFileRingBuffer[E_DB_StructureType.ProductionReport][i](udiNovRamIndex:=i,dataType:=E_DB_StructureType.ProductionReport,NovRamData:=NovRamData);
	fbNovRamToFileRingBuffer[E_DB_StructureType.ProductionSummary][i](udiNovRamIndex:=i,dataType:=E_DB_StructureType.ProductionSummary,NovRamData:=NovRamData);
	fbNovRamToFileRingBuffer[E_DB_StructureType.SoDuration][i](udiNovRamIndex:=i,dataType:=E_DB_StructureType.SoDuration,NovRamData:=NovRamData);
	fbNovRamToFileRingBuffer[E_DB_StructureType.StopCount][i](udiNovRamIndex:=i,dataType:=E_DB_StructureType.StopCount,NovRamData:=NovRamData);
	fbNovRamToFileRingBuffer[E_DB_StructureType.RegularCheckResults][i](udiNovRamIndex:=i,dataType:=E_DB_StructureType.RegularCheckResults,NovRamData:=NovRamData);
	
END_FOR
//File to DB
FOR i:=0 TO gvl.NovRamBufferRatio-1 DO
	FOR k:=0 TO GVL.FileRingBufferRatio-1 DO
		
		fbFileRingBufferToDB[E_DB_StructureType.AlarmHistory][i][k](udiNovRam_BufferIndex:=i,udiFile_Index:=k,dataType:=E_DB_StructureType.AlarmHistory,NovRamData:=NovRamData);
		fbFileRingBufferToDB[E_DB_StructureType.ProductionHistory][i][k](udiNovRam_BufferIndex:=i,udiFile_Index:=k,dataType:=E_DB_StructureType.ProductionHistory,NovRamData:=NovRamData);
		fbFileRingBufferToDB[E_DB_StructureType.ProductionReport][i][k](udiNovRam_BufferIndex:=i,udiFile_Index:=k,dataType:=E_DB_StructureType.ProductionReport,NovRamData:=NovRamData);
		fbFileRingBufferToDB[E_DB_StructureType.ProductionSummary][i][k](udiNovRam_BufferIndex:=i,udiFile_Index:=k,dataType:=E_DB_StructureType.ProductionSummary,NovRamData:=NovRamData);
		fbFileRingBufferToDB[E_DB_StructureType.SoDuration][i][k](udiNovRam_BufferIndex:=i,udiFile_Index:=k,dataType:=E_DB_StructureType.SoDuration,NovRamData:=NovRamData);
		fbFileRingBufferToDB[E_DB_StructureType.StopCount][i][k](udiNovRam_BufferIndex:=i,udiFile_Index:=k,dataType:=E_DB_StructureType.StopCount,NovRamData:=NovRamData);
		fbFileRingBufferToDB[E_DB_StructureType.RegularCheckResults][i][k](udiNovRam_BufferIndex:=i,udiFile_Index:=k,dataType:=E_DB_StructureType.RegularCheckResults,NovRamData:=NovRamData);
		
	END_FOR
END_FOR
END_METHOD

END_FUNCTION_BLOCK

// ---- POUs/DataFlow/Lv2/FB_DataToNovRam.TcPOU
FUNCTION_BLOCK FB_DataToNovRam
VAR_INPUT
	bExecute:BOOL;
	
	savedData:ST_AlarmInfo_DB_save;
END_VAR
VAR_OUTPUT
	bResult:BOOL;
END_VAR
VAR
	
END_VAR
VAR_IN_OUT
	NovRamData:ST_NovRam;
END_VAR

METHOD M_AlarmHistory : BOOL
VAR_INPUT
	addData:ST_AlarmInfo_DB;
END_VAR
VAR
	eStrIndex:DINT;
	udiNowRowIndex:DINT;
	udiWritenIndex:DINT;
	CompressedData:ST_AlarmInfo_DB_save;
END_VAR
//Config
eStrIndex:=E_DB_StructureType.AlarmHistory;
udiNowRowIndex:=NovRamData.arrNovRam_Status[eStrIndex].nowRowIndex;
udiWritenIndex:=NovRamData.arrNovRam_Status[eStrIndex].writenIndex;

IF NovRamData.arrNovRam_Status[eStrIndex].RowDataLocked[udiNowRowIndex]=FALSE THEN//writable
	
	//write data
	M_ST_AlarmHistory_Compress(Input:=addData,Output=>NovRamData.AlarmHistory[udiNowRowIndex][udiWritenIndex]);
	
	NovRamData.arrNovRam_Status[eStrIndex].writenIndex:=NovRamData.arrNovRam_Status[eStrIndex].writenIndex+1;
	
	//Check if Full
	IF NovRamData.arrNovRam_Status[eStrIndex].writenIndex >= (GVL.arrArrayLength[eStrIndex]) THEN
		//Set Row Lock
		NovRamData.arrNovRam_Status[eStrIndex].RowDataLocked[udiNowRowIndex]:=TRUE;
		
		//Reset Row and writenIndex
		NovRamData.arrNovRam_Status[eStrIndex].nowRowIndex:=(udiNowRowIndex+1)MOD GVL.NovRamBufferRatio;
		NovRamData.arrNovRam_Status[eStrIndex].writenIndex:=0;
	END_IF
	
	M_AlarmHistory:=TRUE;
ELSE
	M_AlarmHistory:=FALSE;
END_IF
END_METHOD

METHOD M_ProductionHistory : BOOL
VAR_INPUT
	addData:ST_PHI_GroupData_DB;
END_VAR
VAR 
	eStrIndex:DINT;
	udiNowRowIndex:DINT;
	udiWritenIndex:DINT;
	CompressedData:ST_PHI_GroupData_DB;
END_VAR
//Config
eStrIndex:=E_DB_StructureType.ProductionHistory;
udiNowRowIndex:=NovRamData.arrNovRam_Status[eStrIndex].nowRowIndex;
udiWritenIndex:=NovRamData.arrNovRam_Status[eStrIndex].writenIndex;

IF NovRamData.arrNovRam_Status[eStrIndex].RowDataLocked[udiNowRowIndex]=FALSE THEN//writable
	
	//write data
	M_ST_ProductionHistory_Compress(Input:=addData,Output=>NovRamData.ProductionHistory[udiNowRowIndex][udiWritenIndex]);
	
	NovRamData.arrNovRam_Status[eStrIndex].writenIndex:=NovRamData.arrNovRam_Status[eStrIndex].writenIndex+1;
	
	//Check if Full
	IF NovRamData.arrNovRam_Status[eStrIndex].writenIndex >= (GVL.arrArrayLength[eStrIndex]) THEN
		//Set Row Lock
		NovRamData.arrNovRam_Status[eStrIndex].RowDataLocked[udiNowRowIndex]:=TRUE;
		
		//Reset Row and writenIndex
		NovRamData.arrNovRam_Status[eStrIndex].nowRowIndex:=(udiNowRowIndex+1)MOD GVL.NovRamBufferRatio;
		NovRamData.arrNovRam_Status[eStrIndex].writenIndex:=0;
	END_IF
	
	M_ProductionHistory:=TRUE;
ELSE
	M_ProductionHistory:=FALSE;
END_IF
END_METHOD

METHOD M_ProductionReport : BOOL
VAR_INPUT
	addData:ST_OEE_ProductionReport;
END_VAR
VAR
	eStrIndex:DINT;
	udiNowRowIndex:DINT;
	udiWritenIndex:DINT;
	CompressedData:ST_OEE_ProductionReport;
END_VAR
//Config
eStrIndex:=E_DB_StructureType.ProductionReport;
udiNowRowIndex:=NovRamData.arrNovRam_Status[eStrIndex].nowRowIndex;
udiWritenIndex:=NovRamData.arrNovRam_Status[eStrIndex].writenIndex;

IF NovRamData.arrNovRam_Status[eStrIndex].RowDataLocked[udiNowRowIndex]=FALSE THEN//writable
	
	//write data
	M_ST_ProductionReport_Compress(Input:=addData,Output=>NovRamData.ProductionReport[udiNowRowIndex][udiWritenIndex]);

	NovRamData.arrNovRam_Status[eStrIndex].writenIndex:=NovRamData.arrNovRam_Status[eStrIndex].writenIndex+1;
	
	//Check if Full
	IF NovRamData.arrNovRam_Status[eStrIndex].writenIndex >= (GVL.arrArrayLength[eStrIndex]) THEN
		//Set Row Lock
		NovRamData.arrNovRam_Status[eStrIndex].RowDataLocked[udiNowRowIndex]:=TRUE;
		
		//Reset Row and writenIndex
		NovRamData.arrNovRam_Status[eStrIndex].nowRowIndex:=(udiNowRowIndex+1)MOD GVL.NovRamBufferRatio;
		NovRamData.arrNovRam_Status[eStrIndex].writenIndex:=0;
	END_IF
	
	M_ProductionReport:=TRUE;
ELSE
	M_ProductionReport:=FALSE;
END_IF
END_METHOD

METHOD M_ProductionSummary : BOOL
VAR_INPUT
	addData:ST_OEE_ProductionSummary;
END_VAR
VAR
	eStrIndex:DINT;
	udiNowRowIndex:DINT;
	udiWritenIndex:DINT;
	CompressedData:ST_OEE_ProductionSummary;
END_VAR
//Config
eStrIndex:=E_DB_StructureType.ProductionSummary;
udiNowRowIndex:=NovRamData.arrNovRam_Status[eStrIndex].nowRowIndex;
udiWritenIndex:=NovRamData.arrNovRam_Status[eStrIndex].writenIndex;

IF NovRamData.arrNovRam_Status[eStrIndex].RowDataLocked[udiNowRowIndex]=FALSE THEN//writable
	
	//write data
	M_ST_ProductionSummary_Compress(Input:=addData,Output=>NovRamData.ProductionSummary[udiNowRowIndex][udiWritenIndex]);

	NovRamData.arrNovRam_Status[eStrIndex].writenIndex:=NovRamData.arrNovRam_Status[eStrIndex].writenIndex+1;
	
	//Check if Full
	IF NovRamData.arrNovRam_Status[eStrIndex].writenIndex >= (GVL.arrArrayLength[eStrIndex]) THEN
		//Set Row Lock
		NovRamData.arrNovRam_Status[eStrIndex].RowDataLocked[udiNowRowIndex]:=TRUE;
		
		//Reset Row and writenIndex
		NovRamData.arrNovRam_Status[eStrIndex].nowRowIndex:=(udiNowRowIndex+1)MOD GVL.NovRamBufferRatio;
		NovRamData.arrNovRam_Status[eStrIndex].writenIndex:=0;
	END_IF
	
	M_ProductionSummary:=TRUE;
ELSE
	M_ProductionSummary:=FALSE;
END_IF
END_METHOD

METHOD M_RegularCheckResults : BOOL
VAR_INPUT
	addData:ST_RegularCheck_Results;
END_VAR
VAR
	eStrIndex:DINT;
	udiNowRowIndex:DINT;
	udiWritenIndex:DINT;
	CompressedData:ST_RegularCheck_Results;
END_VAR
//Config
eStrIndex:=E_DB_StructureType.RegularCheckResults;
udiNowRowIndex:=NovRamData.arrNovRam_Status[eStrIndex].nowRowIndex;
udiWritenIndex:=NovRamData.arrNovRam_Status[eStrIndex].writenIndex;

IF NovRamData.arrNovRam_Status[eStrIndex].RowDataLocked[udiNowRowIndex]=FALSE THEN//writable
	
	//write data
	M_ST_RegularCheckResults_Compress(Input:=addData,Output=>NovRamData.RegularCheckResults[udiNowRowIndex][udiWritenIndex]);
	
	NovRamData.arrNovRam_Status[eStrIndex].writenIndex:=NovRamData.arrNovRam_Status[eStrIndex].writenIndex+1;
	
	//Check if Full
	IF NovRamData.arrNovRam_Status[eStrIndex].writenIndex >= (GVL.arrArrayLength[eStrIndex]) THEN
		//Set Row Lock
		NovRamData.arrNovRam_Status[eStrIndex].RowDataLocked[udiNowRowIndex]:=TRUE;
		
		//Reset Row and writenIndex
		NovRamData.arrNovRam_Status[eStrIndex].nowRowIndex:=(udiNowRowIndex+1)MOD GVL.NovRamBufferRatio;
		NovRamData.arrNovRam_Status[eStrIndex].writenIndex:=0;
	END_IF
	
	M_RegularCheckResults:=TRUE;
ELSE
	M_RegularCheckResults:=FALSE;
END_IF
END_METHOD

METHOD M_SoDuration : BOOL
VAR_INPUT
	addData:ST_SoDuration;
END_VAR
VAR
	eStrIndex:DINT;
	udiNowRowIndex:DINT;
	udiWritenIndex:DINT;
	CompressedData:ST_SoDuration;
END_VAR
//Config
eStrIndex:=E_DB_StructureType.SoDuration;
udiNowRowIndex:=NovRamData.arrNovRam_Status[eStrIndex].nowRowIndex;
udiWritenIndex:=NovRamData.arrNovRam_Status[eStrIndex].writenIndex;

IF NovRamData.arrNovRam_Status[eStrIndex].RowDataLocked[udiNowRowIndex]=FALSE THEN//writable
	
	//write data
	M_ST_SoDuration_Compress(Input:=addData,Output=>NovRamData.SoDuration[udiNowRowIndex][udiWritenIndex]);
	
	NovRamData.arrNovRam_Status[eStrIndex].writenIndex:=NovRamData.arrNovRam_Status[eStrIndex].writenIndex+1;
	
	//Check if Full
	IF NovRamData.arrNovRam_Status[eStrIndex].writenIndex >= (GVL.arrArrayLength[eStrIndex]) THEN
		//Set Row Lock
		NovRamData.arrNovRam_Status[eStrIndex].RowDataLocked[udiNowRowIndex]:=TRUE;
		
		//Reset Row and writenIndex
		NovRamData.arrNovRam_Status[eStrIndex].nowRowIndex:=(udiNowRowIndex+1)MOD GVL.NovRamBufferRatio;
		NovRamData.arrNovRam_Status[eStrIndex].writenIndex:=0;
	END_IF
	
	M_SoDuration:=TRUE;
ELSE
	M_SoDuration:=FALSE;
END_IF
END_METHOD

METHOD M_ST_AlarmHistory_Compress : BOOL
VAR_INPUT
	Input:ST_AlarmInfo_DB;
END_VAR
VAR_OUTPUT
	Output:ST_AlarmInfo_DB_save;
END_VAR
Output.lrTime_ms:=Input.lrTime_ms;
Output.iMsgProc:=Input.iMsgProc;
Output.iStateAfter:=Input.iStateAfter;
Output.iMsgClass:=Input.iMsgClass;
Output.diMsgNumber:=Input.diMsgNumber;
Output.sTimeString:=Input.sTimeString;
Output.wsMsgText:=Input.wsMsgText;
Output.sPLC:=Input.sPLC;
Output.wsEquipment:=Input.wsEquipment;
Output.sFaam_id:=Input.sFaam_id;
END_METHOD

METHOD M_ST_ProductionHistory_Compress : BOOL
VAR_INPUT
	Input:ST_PHI_GroupData_DB;
END_VAR
VAR_OUTPUT
	Output:ST_PHI_GroupData_DB;
END_VAR
Output:=Input;
END_METHOD

METHOD M_ST_ProductionReport_Compress : BOOL
VAR_INPUT
	Input:ST_OEE_ProductionReport;
END_VAR
VAR_OUTPUT
	Output:ST_OEE_ProductionReport;
END_VAR
Output:=Input;
END_METHOD

METHOD M_ST_ProductionSummary_Compress : BOOL
VAR_INPUT
	Input:ST_OEE_ProductionSummary;
END_VAR
VAR_OUTPUT
	Output:ST_OEE_ProductionSummary;
END_VAR
Output:=Input;
END_METHOD

METHOD M_ST_RegularCheckResults_Compress : BOOL
VAR_INPUT
	Input:ST_RegularCheck_Results;
END_VAR
VAR_OUTPUT
	Output:ST_RegularCheck_Results;
END_VAR
(*
Output.stProductHistory.diStation_number:=Input.stProductHistory.diStation_number;
Output.stProductHistory.diTrack_number:=Input.stProductHistory.diTrack_number;
Output.stProductHistory.dtStart_time:=Input.stProductHistory.dtStart_time;

IF Input.bSensor = TRUE THEN
	Output.eSensor:=E_RegularCheckSensorResult.Pass;
ELSE
	Output.eSensor:=E_RegularCheckSensorResult.Fail;
END_IF

IF Input.bCamera = TRUE THEN
	Output.eCamera:=E_RegularCheckSensorResult.Pass;
ELSE
	Output.eCamera:=E_RegularCheckSensorResult.Fail;
END_IF

IF Input.bLoadcell = TRUE THEN
	Output.eLoadcell:=E_RegularCheckSensorResult.Pass;
ELSE
	Output.eLoadcell:=E_RegularCheckSensorResult.Fail;
END_IF

IF Input.bSensor2 = TRUE THEN
	Output.eSensor2:=E_RegularCheckSensorResult.Pass;
ELSE
	Output.eSensor2:=E_RegularCheckSensorResult.Fail;
END_IF

Output.diRegular_check_id:=Input.diRegular_check_id;
Output.sFaam_id:=Input.sFaam_id;
Output.sSo_number:=Input.sSo_number;
Output.diSo_id:=Input.diSo_id;
Output.wsEmployee_name_logged_in:=Input.wsEmployee_name_logged_in;
*)
Output:=Input;
END_METHOD

METHOD M_ST_SoDuration_Compress : BOOL
VAR_INPUT
	Input:ST_SoDuration;
END_VAR
VAR_OUTPUT
	Output:ST_SoDuration;
END_VAR
Output:=Input;
END_METHOD

METHOD M_ST_StopCount_Compress : BOOL
VAR_INPUT
	Input:ST_StopCount;
END_VAR
VAR_OUTPUT
	Output:ST_StopCount;
END_VAR
Output:=Input;
END_METHOD

METHOD M_StopCount : BOOL
VAR_INPUT
	addData:ST_StopCount;
END_VAR
VAR
	eStrIndex:DINT;
	udiNowRowIndex:DINT;
	udiWritenIndex:DINT;
	CompressedData:ST_StopCount;
END_VAR
//Config
eStrIndex:=E_DB_StructureType.StopCount;
udiNowRowIndex:=NovRamData.arrNovRam_Status[eStrIndex].nowRowIndex;
udiWritenIndex:=NovRamData.arrNovRam_Status[eStrIndex].writenIndex;

IF NovRamData.arrNovRam_Status[eStrIndex].RowDataLocked[udiNowRowIndex]=FALSE THEN//writable
	
	//write data
	M_ST_StopCount_Compress(Input:=addData,Output=>NovRamData.StopCount[udiNowRowIndex][udiWritenIndex]);

	NovRamData.arrNovRam_Status[eStrIndex].writenIndex:=NovRamData.arrNovRam_Status[eStrIndex].writenIndex+1;
	
	//Check if Full
	IF NovRamData.arrNovRam_Status[eStrIndex].writenIndex >= (GVL.arrArrayLength[eStrIndex]) THEN
		//Set Row Lock
		NovRamData.arrNovRam_Status[eStrIndex].RowDataLocked[udiNowRowIndex]:=TRUE;
		
		//Reset Row and writenIndex
		NovRamData.arrNovRam_Status[eStrIndex].nowRowIndex:=(udiNowRowIndex+1)MOD GVL.NovRamBufferRatio;
		NovRamData.arrNovRam_Status[eStrIndex].writenIndex:=0;
	END_IF
	
	M_StopCount:=TRUE;
ELSE
	M_StopCount:=FALSE;
END_IF
END_METHOD

END_FUNCTION_BLOCK

// ---- POUs/DataFlow/Lv2/FB_NovRamToFileRingBuffer.TcPOU
FUNCTION_BLOCK FB_NovRamToFileRingBuffer
VAR_INPUT
	udiNovRamIndex:UDINT;
	dataType:DINT;
END_VAR
VAR_OUTPUT
	//readData:ARRAY [0..GVL.arrArrayLength[E_DB_StructureType.AlarmHistory]-1] OF ST_AlarmInfo_DB_save;
END_VAR
VAR
	udiVAr1: UDINT;
END_VAR
VAR_IN_OUT
	NovRamData:ST_NovRam;
END_VAR

IF dataType = E_DB_StructureType.AlarmHistory THEN
	M_AlarmHistory(udiNovRamIndex:=udiNovRamIndex);
ELSIF dataType = E_DB_StructureType.ProductionHistory THEN
	M_ProductionHistory(udiNovRamIndex:=udiNovRamIndex);
ELSIF dataType = E_DB_StructureType.ProductionReport THEN
	M_ProductionReport(udiNovRamIndex:=udiNovRamIndex);
ELSIF dataType = E_DB_StructureType.ProductionSummary THEN
	M_ProductionSummary(udiNovRamIndex:=udiNovRamIndex);
ELSIF dataType = E_DB_StructureType.SoDuration THEN
	M_SoDuration(udiNovRamIndex:=udiNovRamIndex);
ELSIF dataType = E_DB_StructureType.StopCount THEN
	M_StopCount(udiNovRamIndex:=udiNovRamIndex);
ELSIF dataType = E_DB_StructureType.RegularCheckResults THEN
	M_RegularCheckResults(udiNovRamIndex:=udiNovRamIndex);
END_IF

METHOD M_AlarmHistory : BOOL
VAR_INPUT
	udiNovRamIndex:UDINT;
END_VAR
VAR_OUTPUT
	
END_VAR
VAR_INST
	WriteData:ARRAY[0..GVL.arrArrayLength[E_DB_StructureType.AlarmHistory]-1] OF ST_AlarmInfo_DB_save;//small
	iStep:INT;
	i:UDINT;
	fbFileRingBuffer: FB_FileRingBuffer := ( sNetId     := '',
                                             sPathName  := '',
                                             ePath      := PATH_GENERIC,
                                             nID        := 1,
                                             cbBuffer   := gvl.arrFileRingBufferSize[E_DB_StructureType.AlarmHistory], //5MB(5*10^6Bytes)
                                             bOverwrite := FALSE,
                                             pWriteBuff := 0,
                                             cbWriteLen := 0,
                                             pReadBuff  := 0,
                                             cbReadLen  := 0,
                                             tTimeout   := T#1S );
	bBusy:BOOL;
	bError:BOOL;
	nErrID:UDINT;
	stHeader:ST_FileRBufferHead;
    loadData  : ARRAY[0..511] OF BYTE :=[512(0)];
    cbLoad    : UDINT;
	
	fileName:STRING(255);
	tempFileIndex:UDINT;
	eStrIndex:DINT;
	
	//1217
	TransTrig:TON;
END_VAR
//Config	
eStrIndex:=E_DB_StructureType.AlarmHistory;

fbFileRingBuffer(sPathName:=fileName
				,bBusy=>bBusy,bError=>bError,nErrID=>nErrID
				,cbReturn=>cbLoad,stHeader=>stHeader);
//1217				
TransTrig(PT:=T#10S);//10s upload one time

CASE iStep OF
	0://NovRam full detect / file full detect
		
		tempFileIndex:=NovRamData.arrFileRingBuffer_Status[eStrIndex].nowFileIndex[udiNovRamIndex];
		
		//1217
		IF NovRamData.arrNovRam_Status[eStrIndex].RowDataLocked[udiNovRamIndex] = FALSE//not full and 
		AND NovRamData.arrNovRam_Status[eStrIndex].writenIndex > 0 THEN//has been writen
			
			TransTrig(IN:=TRUE);
			
			IF TransTrig.Q //timeout
			AND NovRamData.arrFileRingBuffer_Status[eStrIndex].bFileFull[udiNovRamIndex][tempFileIndex] = FALSE THEN//File can write
				TransTrig(IN:=FALSE);
				
				//Set Row Lock
				NovRamData.arrNovRam_Status[eStrIndex].RowDataLocked[udiNovRamIndex]:=TRUE;
				
				//save writen count
				NovRamData.arrNovRam_Status[eStrIndex].writenCount := NovRamData.arrNovRam_Status[eStrIndex].writenIndex;
				
				//Reset Row and writenIndex
				NovRamData.arrNovRam_Status[eStrIndex].nowRowIndex:=(udiNovRamIndex+1)MOD GVL.NovRamBufferRatio;
				NovRamData.arrNovRam_Status[eStrIndex].writenIndex:=0;
		
				fileName:=M_GetFileName(structureType:=eStrIndex
										,udiNovRam_BufferIndex:=udiNovRamIndex
										,udiFile_Index:=NovRamData.arrFileRingBuffer_Status[eStrIndex].nowFileIndex[udiNovRamIndex]);
										
				iStep:=1;
			END_IF
			
		ELSE
			IF NovRamData.arrNovRam_Status[eStrIndex].RowDataLocked[udiNovRamIndex] //NovRam full = should work
			AND NovRamData.arrFileRingBuffer_Status[eStrIndex].bFileFull[udiNovRamIndex][tempFileIndex] = FALSE//File can write
			THEN
				
				//1217
				TransTrig(IN:=FALSE);
				//save writen count
				NovRamData.arrNovRam_Status[eStrIndex].writenCount :=GVL.arrArrayLength[eStrIndex];
				
				fileName:=M_GetFileName(structureType:=eStrIndex
										,udiNovRam_BufferIndex:=udiNovRamIndex
										,udiFile_Index:=NovRamData.arrFileRingBuffer_Status[eStrIndex].nowFileIndex[udiNovRamIndex]);
										
				iStep:=1;
			END_IF
		END_IF
		
		

	1://Open File
		
		fbFileRingBuffer.A_Open();
		
		iStep:=2;
		
	2://Wait Done/Add Data
		IF fbFileRingBuffer.bBusy=FALSE AND NOT fbFileRingBuffer.bError THEN
			//1217
			udiVAr1 := NovRamData.arrNovRam_Status[eStrIndex].writenCount-1;
			//FOR i:=0 TO GVL.arrArrayLength[E_DB_StructureType.AlarmHistory]-1 DO 
			FOR i:=0 TO udiVAr1 DO
				WriteData[i] := NovRamData.AlarmHistory[udiNovRamIndex][i];
			END_FOR
			
			//1217
			//Add
			//fbFileRingBuffer.A_AddTail( pWriteBuff := ADR(WriteData), cbWriteLen := SIZEOF(WriteData),
			//		pReadBuff := 0, cbReadLen:=0 );
			fbFileRingBuffer.A_AddTail( pWriteBuff := ADR(WriteData), cbWriteLen := NovRamData.arrNovRam_Status[eStrIndex].writenCount * SIZEOF(ST_AlarmInfo_DB_save),
					pReadBuff := 0, cbReadLen:=0 );
					
			iStep:=3;
			
		END_IF
	3://Wait Done / Close file /(Check if file Full)
		IF fbFileRingBuffer.bBusy=FALSE THEN
						
			//Check if file full
			IF NOT fbFileRingBuffer.bError THEN
				iStep:=4;
			ELSIF fbFileRingBuffer.bError = TRUE AND nErrID=32768 THEN//full
				iStep:=11;
			END_IF
			
			//close file
			fbFileRingBuffer.A_Close();
			
		END_IF
	4://Wait Done(file still has space)
		IF fbFileRingBuffer.bBusy=FALSE AND NOT fbFileRingBuffer.bError THEN
			
			NovRamData.arrNovRam_Status[eStrIndex].RowDataLocked[udiNovRamIndex]:=FALSE;
			
			iStep:=0;
		END_IF
	11://Wait Done(file full)
		IF fbFileRingBuffer.bBusy=FALSE AND NOT fbFileRingBuffer.bError THEN
			
			//Lock now file
			//NovRamData.arrFileRingBuffer_Status.bFileFull[(gvl.FileRingBufferRatio * udiNovRamIndex) + NovRamData.arrFileRingBuffer_Status.nowFileIndex[udiNovRamIndex]]:=TRUE;
			tempFileIndex:=NovRamData.arrFileRingBuffer_Status[eStrIndex].nowFileIndex[udiNovRamIndex];
			NovRamData.arrFileRingBuffer_Status[eStrIndex].bFileFull[udiNovRamIndex][tempFileIndex]:=TRUE;
			
			//Move to next FileIndex
			NovRamData.arrFileRingBuffer_Status[eStrIndex].nowFileIndex[udiNovRamIndex]:=((NovRamData.arrFileRingBuffer_Status[eStrIndex].nowFileIndex[udiNovRamIndex]+1) MOD GVL.FileRingBufferRatio);
			
			iStep:=0;
			
		END_IF
END_CASE
END_METHOD

METHOD M_GetFileName : STRING(255)
VAR_INPUT
	structureType:DINT;
	udiNovRam_BufferIndex:UDINT;
	udiFile_Index:UDINT;
END_VAR
VAR
	tempString:STRING(255);
	tempString2:STRING(255);
	tempFileNo:UDINT;
END_VAR
IF structureType=E_DB_StructureType.AlarmHistory THEN
	tempString:=CONCAT(gvl.arrfileFolder[structureType],'AlarmHistory');
ELSIF structureType=E_DB_StructureType.ProductionHistory THEN
	tempString:=CONCAT(gvl.arrfileFolder[structureType],'ProductionHistory');
ELSIF structureType=E_DB_StructureType.ProductionReport THEN
	tempString:=CONCAT(gvl.arrfileFolder[structureType],'ProductionReport');
ELSIF structureType=E_DB_StructureType.ProductionSummary THEN
	tempString:=CONCAT(gvl.arrfileFolder[structureType],'ProductionSummary');
ELSIF structureType=E_DB_StructureType.SoDuration THEN
	tempString:=CONCAT(gvl.arrfileFolder[structureType],'SoDuration');
ELSIF structureType=E_DB_StructureType.StopCount THEN
	tempString:=CONCAT(gvl.arrfileFolder[structureType],'StopCount');
ELSIF structureType=E_DB_StructureType.RegularCheckResults THEN
	tempString:=CONCAT(gvl.arrfileFolder[structureType],'RegularCheckResults');
END_IF

tempFileNo:=(udiNovRam_BufferIndex) * GVL.FileRingBufferRatio + (udiFile_Index + 1);
tempString2:=CONCAT(tempString,UDINT_TO_STRING(tempFileNo));
M_GetFileName:=CONCAT(tempString2,'.dat');
END_METHOD

METHOD M_ProductionHistory : BOOL
VAR_INPUT
	udiNovRamIndex:UDINT;
END_VAR
VAR_INST
	WriteData:ARRAY[0..GVL.arrArrayLength[E_DB_StructureType.ProductionHistory]-1] OF ST_PHI_GroupData_DB;//small
	iStep:INT;
	i:UDINT;
	fbFileRingBuffer: FB_FileRingBuffer := ( sNetId     := '',
                                             sPathName  := '',
                                             ePath      := PATH_GENERIC,
                                             nID        := 1,
                                             cbBuffer   := gvl.arrFileRingBufferSize[E_DB_StructureType.ProductionHistory], //5MB(5*10^6Bytes)
                                             bOverwrite := FALSE,
                                             pWriteBuff := 0,
                                             cbWriteLen := 0,
                                             pReadBuff  := 0,
                                             cbReadLen  := 0,
                                             tTimeout   := T#1S );
	bBusy:BOOL;
	bError:BOOL;
	nErrID:UDINT;
	stHeader:ST_FileRBufferHead;
    loadData  : ARRAY[0..511] OF BYTE :=[512(0)];
    cbLoad    : UDINT;
	
	fileName:STRING(255);
	tempFileIndex:UDINT;
	eStrIndex:DINT;
END_VAR
//Config
eStrIndex:=E_DB_StructureType.ProductionHistory;

fbFileRingBuffer(sPathName:=fileName
				,bBusy=>bBusy,bError=>bError,nErrID=>nErrID
				,cbReturn=>cbLoad,stHeader=>stHeader);

CASE iStep OF
	0://NovRam full detect / file full detect
		
		tempFileIndex:=NovRamData.arrFileRingBuffer_Status[eStrIndex].nowFileIndex[udiNovRamIndex];
		
		IF NovRamData.arrNovRam_Status[eStrIndex].RowDataLocked[udiNovRamIndex] //NovRam full = should work
		AND NovRamData.arrFileRingBuffer_Status[eStrIndex].bFileFull[udiNovRamIndex][tempFileIndex] = FALSE//File can write
		THEN
			//
			fileName:=M_GetFileName(structureType:=eStrIndex
									,udiNovRam_BufferIndex:=udiNovRamIndex
									,udiFile_Index:=NovRamData.arrFileRingBuffer_Status[eStrIndex].nowFileIndex[udiNovRamIndex]);
									
			iStep:=1;
		END_IF

	1://Open File
		
		fbFileRingBuffer.A_Open();
		
		iStep:=2;
		
	2://Wait Done/Add Data
		IF fbFileRingBuffer.bBusy=FALSE AND NOT fbFileRingBuffer.bError THEN
			
			FOR i:=0 TO GVL.arrArrayLength[E_DB_StructureType.ProductionHistory]-1 DO 
				WriteData[i] := NovRamData.ProductionHistory[udiNovRamIndex][i];
			END_FOR
			
			//Add
			fbFileRingBuffer.A_AddTail( pWriteBuff := ADR(WriteData), cbWriteLen := SIZEOF(WriteData),
					pReadBuff := 0, cbReadLen:=0 );
			
			iStep:=3;
			
		END_IF
	3://Wait Done / Close file /(Check if file Full)
		IF fbFileRingBuffer.bBusy=FALSE THEN
						
			//Check if file full
			IF NOT fbFileRingBuffer.bError THEN
				iStep:=4;
			ELSIF fbFileRingBuffer.bError = TRUE AND nErrID=32768 THEN//full
				iStep:=11;
			END_IF
			
			//close file
			fbFileRingBuffer.A_Close();
			
		END_IF
	4://Wait Done(file still has space)
		IF fbFileRingBuffer.bBusy=FALSE AND NOT fbFileRingBuffer.bError THEN
			
			NovRamData.arrNovRam_Status[eStrIndex].RowDataLocked[udiNovRamIndex]:=FALSE;
			
			iStep:=0;
		END_IF
	11://Wait Done(file full)
		IF fbFileRingBuffer.bBusy=FALSE AND NOT fbFileRingBuffer.bError THEN
			
			//Lock now file
			//NovRamData.FileRingBuffer_Status.bFileFull[(gvl.FileRingBufferRatio * udiNovRamIndex) + NovRamData.FileRingBuffer_Status.nowFileIndex[udiNovRamIndex]]:=TRUE;
			tempFileIndex:=NovRamData.arrFileRingBuffer_Status[eStrIndex].nowFileIndex[udiNovRamIndex];
			NovRamData.arrFileRingBuffer_Status[eStrIndex].bFileFull[udiNovRamIndex][tempFileIndex]:=TRUE;
			
			//Move to next FileIndex
			NovRamData.arrFileRingBuffer_Status[eStrIndex].nowFileIndex[udiNovRamIndex]:=((NovRamData.arrFileRingBuffer_Status[eStrIndex].nowFileIndex[udiNovRamIndex]+1) MOD GVL.FileRingBufferRatio);
			
			iStep:=0;
			
		END_IF
END_CASE
END_METHOD

METHOD M_ProductionReport : BOOL
VAR_INPUT
	udiNovRamIndex:UDINT;
END_VAR
VAR_INST
	WriteData:ARRAY[0..GVL.arrArrayLength[E_DB_StructureType.ProductionReport]-1] OF ST_OEE_ProductionReport;//small
	iStep:INT;
	i:UDINT;
	fbFileRingBuffer: FB_FileRingBuffer := ( sNetId     := '',
                                             sPathName  := '',
                                             ePath      := PATH_GENERIC,
                                             nID        := 1,
                                             cbBuffer   := gvl.arrFileRingBufferSize[E_DB_StructureType.ProductionReport], //5MB(5*10^6Bytes)
                                             bOverwrite := FALSE,
                                             pWriteBuff := 0,
                                             cbWriteLen := 0,
                                             pReadBuff  := 0,
                                             cbReadLen  := 0,
                                             tTimeout   := T#1S );
	bBusy:BOOL;
	bError:BOOL;
	nErrID:UDINT;
	stHeader:ST_FileRBufferHead;
    loadData  : ARRAY[0..511] OF BYTE :=[512(0)];
    cbLoad    : UDINT;
	
	fileName:STRING(255);
	tempFileIndex:UDINT;
	eStrIndex:DINT;
END_VAR
//Config
eStrIndex:=E_DB_StructureType.ProductionReport;

fbFileRingBuffer(sPathName:=fileName
				,bBusy=>bBusy,bError=>bError,nErrID=>nErrID
				,cbReturn=>cbLoad,stHeader=>stHeader);

CASE iStep OF
	0://NovRam full detect / file full detect
		
		tempFileIndex:=NovRamData.arrFileRingBuffer_Status[eStrIndex].nowFileIndex[udiNovRamIndex];
		
		IF NovRamData.arrNovRam_Status[eStrIndex].RowDataLocked[udiNovRamIndex] //NovRam full = should work
		AND NovRamData.arrFileRingBuffer_Status[eStrIndex].bFileFull[udiNovRamIndex][tempFileIndex] = FALSE//File can write
		THEN
			//
			fileName:=M_GetFileName(structureType:=eStrIndex
									,udiNovRam_BufferIndex:=udiNovRamIndex
									,udiFile_Index:=NovRamData.arrFileRingBuffer_Status[eStrIndex].nowFileIndex[udiNovRamIndex]);
									
			iStep:=1;
		END_IF

	1://Open File
		
		fbFileRingBuffer.A_Open();
		
		iStep:=2;
		
	2://Wait Done/Add Data
		IF fbFileRingBuffer.bBusy=FALSE AND NOT fbFileRingBuffer.bError THEN
			
			FOR i:=0 TO GVL.arrArrayLength[E_DB_StructureType.ProductionReport]-1 DO 
				WriteData[i] := NovRamData.ProductionReport[udiNovRamIndex][i];
			END_FOR
			
			//Add
			fbFileRingBuffer.A_AddTail( pWriteBuff := ADR(WriteData), cbWriteLen := SIZEOF(WriteData),
					pReadBuff := 0, cbReadLen:=0 );
			
			iStep:=3;
			
		END_IF
	3://Wait Done / Close file /(Check if file Full)
		IF fbFileRingBuffer.bBusy=FALSE THEN
						
			//Check if file full
			IF NOT fbFileRingBuffer.bError THEN
				iStep:=4;
			ELSIF fbFileRingBuffer.bError = TRUE AND nErrID=32768 THEN//full
				iStep:=11;
			END_IF
			
			//close file
			fbFileRingBuffer.A_Close();
			
		END_IF
	4://Wait Done(file still has space)
		IF fbFileRingBuffer.bBusy=FALSE AND NOT fbFileRingBuffer.bError THEN
			
			NovRamData.arrNovRam_Status[eStrIndex].RowDataLocked[udiNovRamIndex]:=FALSE;
			
			iStep:=0;
		END_IF
	11://Wait Done(file full)
		IF fbFileRingBuffer.bBusy=FALSE AND NOT fbFileRingBuffer.bError THEN
			
			//Lock now file
			//NovRamData.FileRingBuffer_Status.bFileFull[(gvl.FileRingBufferRatio * udiNovRamIndex) + NovRamData.FileRingBuffer_Status.nowFileIndex[udiNovRamIndex]]:=TRUE;
			tempFileIndex:=NovRamData.arrFileRingBuffer_Status[eStrIndex].nowFileIndex[udiNovRamIndex];
			NovRamData.arrFileRingBuffer_Status[eStrIndex].bFileFull[udiNovRamIndex][tempFileIndex]:=TRUE;
			
			//Move to next FileIndex
			NovRamData.arrFileRingBuffer_Status[eStrIndex].nowFileIndex[udiNovRamIndex]:=((NovRamData.arrFileRingBuffer_Status[eStrIndex].nowFileIndex[udiNovRamIndex]+1) MOD GVL.FileRingBufferRatio);
			
			iStep:=0;
			
		END_IF
END_CASE
END_METHOD

METHOD M_ProductionSummary : BOOL
VAR_INPUT
	udiNovRamIndex:UDINT;
END_VAR
VAR_INST
	WriteData:ARRAY[0..GVL.arrArrayLength[E_DB_StructureType.ProductionSummary]-1] OF ST_OEE_ProductionSummary;//small
	iStep:INT;
	i:UDINT;
	fbFileRingBuffer: FB_FileRingBuffer := ( sNetId     := '',
                                             sPathName  := '',
                                             ePath      := PATH_GENERIC,
                                             nID        := 1,
                                             cbBuffer   := gvl.arrFileRingBufferSize[E_DB_StructureType.ProductionSummary], //5MB(5*10^6Bytes)
                                             bOverwrite := FALSE,
                                             pWriteBuff := 0,
                                             cbWriteLen := 0,
                                             pReadBuff  := 0,
                                             cbReadLen  := 0,
                                             tTimeout   := T#1S );
	bBusy:BOOL;
	bError:BOOL;
	nErrID:UDINT;
	stHeader:ST_FileRBufferHead;
    loadData  : ARRAY[0..511] OF BYTE :=[512(0)];
    cbLoad    : UDINT;
	
	fileName:STRING(255);
	tempFileIndex:UDINT;
	eStrIndex:DINT;
END_VAR
//Config
eStrIndex:=E_DB_StructureType.ProductionSummary;

fbFileRingBuffer(sPathName:=fileName
				,bBusy=>bBusy,bError=>bError,nErrID=>nErrID
				,cbReturn=>cbLoad,stHeader=>stHeader);

CASE iStep OF
	0://NovRam full detect / file full detect
		
		tempFileIndex:=NovRamData.arrFileRingBuffer_Status[eStrIndex].nowFileIndex[udiNovRamIndex];
		
		IF NovRamData.arrNovRam_Status[eStrIndex].RowDataLocked[udiNovRamIndex] //NovRam full = should work
		AND NovRamData.arrFileRingBuffer_Status[eStrIndex].bFileFull[udiNovRamIndex][tempFileIndex] = FALSE//File can write
		THEN
			//
			fileName:=M_GetFileName(structureType:=eStrIndex
									,udiNovRam_BufferIndex:=udiNovRamIndex
									,udiFile_Index:=NovRamData.arrFileRingBuffer_Status[eStrIndex].nowFileIndex[udiNovRamIndex]);
									
			iStep:=1;
		END_IF

	1://Open File
		
		fbFileRingBuffer.A_Open();
		
		iStep:=2;
		
	2://Wait Done/Add Data
		IF fbFileRingBuffer.bBusy=FALSE AND NOT fbFileRingBuffer.bError THEN
			
			FOR i:=0 TO GVL.arrArrayLength[E_DB_StructureType.ProductionSummary]-1 DO 
				WriteData[i] := NovRamData.ProductionSummary[udiNovRamIndex][i];
			END_FOR
			
			//Add
			fbFileRingBuffer.A_AddTail( pWriteBuff := ADR(WriteData), cbWriteLen := SIZEOF(WriteData),
					pReadBuff := 0, cbReadLen:=0 );
			
			iStep:=3;
			
		END_IF
	3://Wait Done / Close file /(Check if file Full)
		IF fbFileRingBuffer.bBusy=FALSE THEN
						
			//Check if file full
			IF NOT fbFileRingBuffer.bError THEN
				iStep:=4;
			ELSIF fbFileRingBuffer.bError = TRUE AND nErrID=32768 THEN//full
				iStep:=11;
			END_IF
			
			//close file
			fbFileRingBuffer.A_Close();
			
		END_IF
	4://Wait Done(file still has space)
		IF fbFileRingBuffer.bBusy=FALSE AND NOT fbFileRingBuffer.bError THEN
			
			NovRamData.arrNovRam_Status[eStrIndex].RowDataLocked[udiNovRamIndex]:=FALSE;
			
			iStep:=0;
		END_IF
	11://Wait Done(file full)
		IF fbFileRingBuffer.bBusy=FALSE AND NOT fbFileRingBuffer.bError THEN
			
			//Lock now file
			//NovRamData.FileRingBuffer_Status.bFileFull[(gvl.FileRingBufferRatio * udiNovRamIndex) + NovRamData.FileRingBuffer_Status.nowFileIndex[udiNovRamIndex]]:=TRUE;
			tempFileIndex:=NovRamData.arrFileRingBuffer_Status[eStrIndex].nowFileIndex[udiNovRamIndex];
			NovRamData.arrFileRingBuffer_Status[eStrIndex].bFileFull[udiNovRamIndex][tempFileIndex]:=TRUE;
			
			//Move to next FileIndex
			NovRamData.arrFileRingBuffer_Status[eStrIndex].nowFileIndex[udiNovRamIndex]:=((NovRamData.arrFileRingBuffer_Status[eStrIndex].nowFileIndex[udiNovRamIndex]+1) MOD GVL.FileRingBufferRatio);
			
			iStep:=0;
			
		END_IF
END_CASE
END_METHOD

METHOD M_RegularCheckResults : BOOL
VAR_INPUT
	udiNovRamIndex:UDINT;
END_VAR
VAR_INST
	WriteData:ARRAY[0..GVL.arrArrayLength[E_DB_StructureType.RegularCheckResults]-1] OF ST_RegularCheck_Results;//small
	iStep:INT;
	i:UDINT;
	fbFileRingBuffer: FB_FileRingBuffer := ( sNetId     := '',
                                             sPathName  := '',
                                             ePath      := PATH_GENERIC,
                                             nID        := 1,
                                             cbBuffer   := gvl.arrFileRingBufferSize[E_DB_StructureType.RegularCheckResults], //5MB(5*10^6Bytes)
                                             bOverwrite := FALSE,
                                             pWriteBuff := 0,
                                             cbWriteLen := 0,
                                             pReadBuff  := 0,
                                             cbReadLen  := 0,
                                             tTimeout   := T#1S );
	bBusy:BOOL;
	bError:BOOL;
	nErrID:UDINT;
	stHeader:ST_FileRBufferHead;
    loadData  : ARRAY[0..511] OF BYTE :=[512(0)];
    cbLoad    : UDINT;
	
	fileName:STRING(255);
	tempFileIndex:UDINT;
	eStrIndex:DINT;
END_VAR
//Config
eStrIndex:=E_DB_StructureType.RegularCheckResults;

fbFileRingBuffer(sPathName:=fileName
				,bBusy=>bBusy,bError=>bError,nErrID=>nErrID
				,cbReturn=>cbLoad,stHeader=>stHeader);

CASE iStep OF
	0://NovRam full detect / file full detect
		
		tempFileIndex:=NovRamData.arrFileRingBuffer_Status[eStrIndex].nowFileIndex[udiNovRamIndex];
		
		IF NovRamData.arrNovRam_Status[eStrIndex].RowDataLocked[udiNovRamIndex] //NovRam full = should work
		AND NovRamData.arrFileRingBuffer_Status[eStrIndex].bFileFull[udiNovRamIndex][tempFileIndex] = FALSE//File can write
		THEN
			//
			fileName:=M_GetFileName(structureType:=eStrIndex
									,udiNovRam_BufferIndex:=udiNovRamIndex
									,udiFile_Index:=NovRamData.arrFileRingBuffer_Status[eStrIndex].nowFileIndex[udiNovRamIndex]);
									
			iStep:=1;
		END_IF

	1://Open File
		
		fbFileRingBuffer.A_Open();
		
		iStep:=2;
		
	2://Wait Done/Add Data
		IF fbFileRingBuffer.bBusy=FALSE AND NOT fbFileRingBuffer.bError THEN
			
			FOR i:=0 TO GVL.arrArrayLength[E_DB_StructureType.RegularCheckResults]-1 DO 
				WriteData[i] := NovRamData.RegularCheckResults[udiNovRamIndex][i];
			END_FOR
			
			//Add
			fbFileRingBuffer.A_AddTail( pWriteBuff := ADR(WriteData), cbWriteLen := SIZEOF(WriteData),
					pReadBuff := 0, cbReadLen:=0 );
			
			iStep:=3;
			
		END_IF
	3://Wait Done / Close file /(Check if file Full)
		IF fbFileRingBuffer.bBusy=FALSE THEN
						
			//Check if file full
			IF NOT fbFileRingBuffer.bError THEN
				iStep:=4;
			ELSIF fbFileRingBuffer.bError = TRUE AND nErrID=32768 THEN//full
				iStep:=11;
			END_IF
			
			//close file
			fbFileRingBuffer.A_Close();
			
		END_IF
	4://Wait Done(file still has space)
		IF fbFileRingBuffer.bBusy=FALSE AND NOT fbFileRingBuffer.bError THEN
			
			NovRamData.arrNovRam_Status[eStrIndex].RowDataLocked[udiNovRamIndex]:=FALSE;
			
			iStep:=0;
		END_IF
	11://Wait Done(file full)
		IF fbFileRingBuffer.bBusy=FALSE AND NOT fbFileRingBuffer.bError THEN
			
			//Lock now file
			//NovRamData.FileRingBuffer_Status.bFileFull[(gvl.FileRingBufferRatio * udiNovRamIndex) + NovRamData.FileRingBuffer_Status.nowFileIndex[udiNovRamIndex]]:=TRUE;
			tempFileIndex:=NovRamData.arrFileRingBuffer_Status[eStrIndex].nowFileIndex[udiNovRamIndex];
			NovRamData.arrFileRingBuffer_Status[eStrIndex].bFileFull[udiNovRamIndex][tempFileIndex]:=TRUE;
			
			//Move to next FileIndex
			NovRamData.arrFileRingBuffer_Status[eStrIndex].nowFileIndex[udiNovRamIndex]:=((NovRamData.arrFileRingBuffer_Status[eStrIndex].nowFileIndex[udiNovRamIndex]+1) MOD GVL.FileRingBufferRatio);
			
			iStep:=0;
			
		END_IF
END_CASE
END_METHOD

METHOD M_SoDuration : BOOL
VAR_INPUT
	udiNovRamIndex:UDINT;
END_VAR
VAR_INST
	WriteData:ARRAY[0..GVL.arrArrayLength[E_DB_StructureType.SoDuration]-1] OF ST_SoDuration;//small
	iStep:INT;
	i:UDINT;
	fbFileRingBuffer: FB_FileRingBuffer := ( sNetId     := '',
                                             sPathName  := '',
                                             ePath      := PATH_GENERIC,
                                             nID        := 1,
                                             cbBuffer   := gvl.arrFileRingBufferSize[E_DB_StructureType.SoDuration], //5MB(5*10^6Bytes)
                                             bOverwrite := FALSE,
                                             pWriteBuff := 0,
                                             cbWriteLen := 0,
                                             pReadBuff  := 0,
                                             cbReadLen  := 0,
                                             tTimeout   := T#1S );
	bBusy:BOOL;
	bError:BOOL;
	nErrID:UDINT;
	stHeader:ST_FileRBufferHead;
    loadData  : ARRAY[0..511] OF BYTE :=[512(0)];
    cbLoad    : UDINT;
	
	fileName:STRING(255);
	tempFileIndex:UDINT;
	eStrIndex:DINT;
END_VAR
//Config
eStrIndex:=E_DB_StructureType.SoDuration;

fbFileRingBuffer(sPathName:=fileName
				,bBusy=>bBusy,bError=>bError,nErrID=>nErrID
				,cbReturn=>cbLoad,stHeader=>stHeader);

CASE iStep OF
	0://NovRam full detect / file full detect
		
		tempFileIndex:=NovRamData.arrFileRingBuffer_Status[eStrIndex].nowFileIndex[udiNovRamIndex];
		
		IF NovRamData.arrNovRam_Status[eStrIndex].RowDataLocked[udiNovRamIndex] //NovRam full = should work
		AND NovRamData.arrFileRingBuffer_Status[eStrIndex].bFileFull[udiNovRamIndex][tempFileIndex] = FALSE//File can write
		THEN
			//
			fileName:=M_GetFileName(structureType:=eStrIndex
									,udiNovRam_BufferIndex:=udiNovRamIndex
									,udiFile_Index:=NovRamData.arrFileRingBuffer_Status[eStrIndex].nowFileIndex[udiNovRamIndex]);
									
			iStep:=1;
		END_IF

	1://Open File
		
		fbFileRingBuffer.A_Open();
		
		iStep:=2;
		
	2://Wait Done/Add Data
		IF fbFileRingBuffer.bBusy=FALSE AND NOT fbFileRingBuffer.bError THEN
			
			FOR i:=0 TO GVL.arrArrayLength[E_DB_StructureType.SoDuration]-1 DO 
				WriteData[i] := NovRamData.SoDuration[udiNovRamIndex][i];
			END_FOR
			
			//Add
			fbFileRingBuffer.A_AddTail( pWriteBuff := ADR(WriteData), cbWriteLen := SIZEOF(WriteData),
					pReadBuff := 0, cbReadLen:=0 );
			
			iStep:=3;
			
		END_IF
	3://Wait Done / Close file /(Check if file Full)
		IF fbFileRingBuffer.bBusy=FALSE THEN
						
			//Check if file full
			IF NOT fbFileRingBuffer.bError THEN
				iStep:=4;
			ELSIF fbFileRingBuffer.bError = TRUE AND nErrID=32768 THEN//full
				iStep:=11;
			END_IF
			
			//close file
			fbFileRingBuffer.A_Close();
			
		END_IF
	4://Wait Done(file still has space)
		IF fbFileRingBuffer.bBusy=FALSE AND NOT fbFileRingBuffer.bError THEN
			
			NovRamData.arrNovRam_Status[eStrIndex].RowDataLocked[udiNovRamIndex]:=FALSE;
			
			iStep:=0;
		END_IF
	11://Wait Done(file full)
		IF fbFileRingBuffer.bBusy=FALSE AND NOT fbFileRingBuffer.bError THEN
			
			//Lock now file
			//NovRamData.FileRingBuffer_Status.bFileFull[(gvl.FileRingBufferRatio * udiNovRamIndex) + NovRamData.FileRingBuffer_Status.nowFileIndex[udiNovRamIndex]]:=TRUE;
			tempFileIndex:=NovRamData.arrFileRingBuffer_Status[eStrIndex].nowFileIndex[udiNovRamIndex];
			NovRamData.arrFileRingBuffer_Status[eStrIndex].bFileFull[udiNovRamIndex][tempFileIndex]:=TRUE;
			
			//Move to next FileIndex
			NovRamData.arrFileRingBuffer_Status[eStrIndex].nowFileIndex[udiNovRamIndex]:=((NovRamData.arrFileRingBuffer_Status[eStrIndex].nowFileIndex[udiNovRamIndex]+1) MOD GVL.FileRingBufferRatio);
			
			iStep:=0;
			
		END_IF
END_CASE
END_METHOD

METHOD M_StopCount : BOOL
VAR_INPUT
	udiNovRamIndex:UDINT;
END_VAR
VAR_INST
	WriteData:ARRAY[0..GVL.arrArrayLength[E_DB_StructureType.StopCount]-1] OF ST_StopCount;//small
	iStep:INT;
	i:UDINT;
	fbFileRingBuffer: FB_FileRingBuffer := ( sNetId     := '',
                                             sPathName  := '',
                                             ePath      := PATH_GENERIC,
                                             nID        := 1,
                                             cbBuffer   := gvl.arrFileRingBufferSize[E_DB_StructureType.StopCount], //5MB(5*10^6Bytes)
                                             bOverwrite := FALSE,
                                             pWriteBuff := 0,
                                             cbWriteLen := 0,
                                             pReadBuff  := 0,
                                             cbReadLen  := 0,
                                             tTimeout   := T#1S );
	bBusy:BOOL;
	bError:BOOL;
	nErrID:UDINT;
	stHeader:ST_FileRBufferHead;
    loadData  : ARRAY[0..511] OF BYTE :=[512(0)];
    cbLoad    : UDINT;
	
	fileName:STRING(255);
	tempFileIndex:UDINT;
	eStrIndex:DINT;
END_VAR
//Config
eStrIndex:=E_DB_StructureType.StopCount;

fbFileRingBuffer(sPathName:=fileName
				,bBusy=>bBusy,bError=>bError,nErrID=>nErrID
				,cbReturn=>cbLoad,stHeader=>stHeader);

CASE iStep OF
	0://NovRam full detect / file full detect
		
		tempFileIndex:=NovRamData.arrFileRingBuffer_Status[eStrIndex].nowFileIndex[udiNovRamIndex];
		
		IF NovRamData.arrNovRam_Status[eStrIndex].RowDataLocked[udiNovRamIndex] //NovRam full = should work
		AND NovRamData.arrFileRingBuffer_Status[eStrIndex].bFileFull[udiNovRamIndex][tempFileIndex] = FALSE//File can write
		THEN
			//
			fileName:=M_GetFileName(structureType:=eStrIndex
									,udiNovRam_BufferIndex:=udiNovRamIndex
									,udiFile_Index:=NovRamData.arrFileRingBuffer_Status[eStrIndex].nowFileIndex[udiNovRamIndex]);
									
			iStep:=1;
		END_IF

	1://Open File
		
		fbFileRingBuffer.A_Open();
		
		iStep:=2;
		
	2://Wait Done/Add Data
		IF fbFileRingBuffer.bBusy=FALSE AND NOT fbFileRingBuffer.bError THEN
			
			FOR i:=0 TO GVL.arrArrayLength[E_DB_StructureType.StopCount]-1 DO 
				WriteData[i] := NovRamData.StopCount[udiNovRamIndex][i];
			END_FOR
			
			//Add
			fbFileRingBuffer.A_AddTail( pWriteBuff := ADR(WriteData), cbWriteLen := SIZEOF(WriteData),
					pReadBuff := 0, cbReadLen:=0 );
			
			iStep:=3;
			
		END_IF
	3://Wait Done / Close file /(Check if file Full)
		IF fbFileRingBuffer.bBusy=FALSE THEN
						
			//Check if file full
			IF NOT fbFileRingBuffer.bError THEN
				iStep:=4;
			ELSIF fbFileRingBuffer.bError = TRUE AND nErrID=32768 THEN//full
				iStep:=11;
			END_IF
			
			//close file
			fbFileRingBuffer.A_Close();
			
		END_IF
	4://Wait Done(file still has space)
		IF fbFileRingBuffer.bBusy=FALSE AND NOT fbFileRingBuffer.bError THEN
			
			NovRamData.arrNovRam_Status[eStrIndex].RowDataLocked[udiNovRamIndex]:=FALSE;
			
			iStep:=0;
		END_IF
	11://Wait Done(file full)
		IF fbFileRingBuffer.bBusy=FALSE AND NOT fbFileRingBuffer.bError THEN
			
			//Lock now file
			//NovRamData.FileRingBuffer_Status.bFileFull[(gvl.FileRingBufferRatio * udiNovRamIndex) + NovRamData.FileRingBuffer_Status.nowFileIndex[udiNovRamIndex]]:=TRUE;
			tempFileIndex:=NovRamData.arrFileRingBuffer_Status[eStrIndex].nowFileIndex[udiNovRamIndex];
			NovRamData.arrFileRingBuffer_Status[eStrIndex].bFileFull[udiNovRamIndex][tempFileIndex]:=TRUE;
			
			//Move to next FileIndex
			NovRamData.arrFileRingBuffer_Status[eStrIndex].nowFileIndex[udiNovRamIndex]:=((NovRamData.arrFileRingBuffer_Status[eStrIndex].nowFileIndex[udiNovRamIndex]+1) MOD GVL.FileRingBufferRatio);
			
			iStep:=0;
			
		END_IF
END_CASE
END_METHOD

END_FUNCTION_BLOCK

// ---- POUs/DataFlow/Lv2/FB_FileRingBufferToDB.TcPOU
FUNCTION_BLOCK FB_FileRingBufferToDB
VAR_INPUT
	udiNovRam_BufferIndex:UDINT;
	udiFile_Index:UDINT;
	dataType:DINT;
END_VAR
VAR_IN_OUT
	NovRamData:ST_NovRam;
END_VAR
VAR
	fbDataUpload_Leo:FB_DataUpload_Leo;
END_VAR


fbDataUpload_Leo();

IF dataType = E_DB_StructureType.AlarmHistory THEN
	M_AlarmHistory(udiNovRam_BufferIndex:=udiNovRam_BufferIndex,udiFile_Index:=udiFile_Index);
ELSIF dataType = E_DB_StructureType.ProductionHistory THEN
	M_ProductionHistory(udiNovRam_BufferIndex:=udiNovRam_BufferIndex,udiFile_Index:=udiFile_Index);
ELSIF dataType = E_DB_StructureType.ProductionReport THEN
	M_ProductionReport(udiNovRam_BufferIndex:=udiNovRam_BufferIndex,udiFile_Index:=udiFile_Index);
ELSIF dataType = E_DB_StructureType.ProductionSummary THEN
	M_ProductionSummary(udiNovRam_BufferIndex:=udiNovRam_BufferIndex,udiFile_Index:=udiFile_Index);
ELSIF dataType = E_DB_StructureType.SoDuration THEN
	M_SoDuration(udiNovRam_BufferIndex:=udiNovRam_BufferIndex,udiFile_Index:=udiFile_Index);
ELSIF dataType = E_DB_StructureType.StopCount THEN
	M_StopCount(udiNovRam_BufferIndex:=udiNovRam_BufferIndex,udiFile_Index:=udiFile_Index);
ELSIF dataType = E_DB_StructureType.RegularCheckResults THEN
	M_RegularCheckResults(udiNovRam_BufferIndex:=udiNovRam_BufferIndex,udiFile_Index:=udiFile_Index);
END_IF

METHOD M_AlarmHistory : BOOL
VAR_INPUT
	
	//udiFileNo:UDINT;
	udiNovRam_BufferIndex:UDINT;
	udiFile_Index:UDINT;
END_VAR
VAR_INST
	arrDataFromFile:ARRAY[0..GVL.arrArrayLength[E_DB_StructureType.AlarmHistory]-1] OF ST_AlarmInfo_DB_save;//small
	DataToDB:ST_AlarmInfo_DB;//large
	AnalizeIndex:UDINT;//should be kept by NovRam
	iStep:INT;
	i:UDINT;
	fbFileRingBuffer: FB_FileRingBuffer := ( sNetId     := '',
                                             sPathName  := '',
                                             ePath      := PATH_GENERIC,
                                             nID        := 1,
                                             cbBuffer   := gvl.arrFileRingBufferSize[E_DB_StructureType.AlarmHistory], //5MB(5*10^6Bytes)
                                             bOverwrite := FALSE,
                                             pWriteBuff := 0,
                                             cbWriteLen := 0,
                                             pReadBuff  := 0,
                                             cbReadLen  := 0,
                                             tTimeout   := T#1S );
	bBusy:BOOL;
	bError:BOOL;
	nErrID:UDINT;
	stHeader:ST_FileRBufferHead;
    //loadData  : ARRAY[0..511] OF BYTE :=[512(0)];
    //cbLoad    : UDINT;
	
	fileName: STRING(255);
	eStrIndex:DINT;
	fbAlarmHistory_DB		: FB_AlarmHistory_DB;
	
	//1217
	TransTrig:TON;
	tempFileIndex:UDINT;
	udiDataCount:UDINT;
	lrTemp:LREAL;
END_VAR
//Config
eStrIndex:=E_DB_StructureType.AlarmHistory;

fbFileRingBuffer(sPathName:=fileName
				,bBusy=>bBusy,bError=>bError,nErrID=>nErrID
				,stHeader=>stHeader);
//DB_Test
fbAlarmHistory_DB(udiDBID:=1);

TransTrig(PT:=T#20S);

CASE iStep OF
	0://check if file full 
		
		//1217
		tempFileIndex:=NovRamData.arrFileRingBuffer_Status[eStrIndex].nowFileIndex[udiNovRam_BufferIndex];
		IF tempFileIndex = udiFile_Index//now writen file index = myself file index
		AND NovRamData.arrFileRingBuffer_Status[eStrIndex].bFileFull[udiNovRam_BufferIndex][udiFile_Index] = FALSE THEN//file not full
			TransTrig(IN:=TRUE);
			
			IF TransTrig.Q THEN//timeout
				TransTrig(in:=FALSE);
				//force to be full
				NovRamData.arrFileRingBuffer_Status[eStrIndex].bFileFull[udiNovRam_BufferIndex][udiFile_Index] := TRUE;
				
				fileName:=M_GetFileName(structureType:=eStrIndex
										,udiNovRam_BufferIndex:=udiNovRam_BufferIndex
										,udiFile_Index:=udiFile_Index);
				
				iStep:=100;
				
			END_IF
		ELSE
			IF NovRamData.arrFileRingBuffer_Status[eStrIndex].bFileFull[udiNovRam_BufferIndex][udiFile_Index] = TRUE//file full = should work 
			THEN
				//1217
				TransTrig(in:=FALSE);
				fileName:=M_GetFileName(structureType:=eStrIndex
										,udiNovRam_BufferIndex:=udiNovRam_BufferIndex
										,udiFile_Index:=udiFile_Index);
				
				iStep:=100;
			END_IF
		END_IF
		
		
	100:// Open file
		
		AnalizeIndex:=0;
		fbFileRingBuffer.A_Open();
		
		iStep:=200;
	200://wait done / read head
		IF NOT fbFileRingBuffer.bBusy AND NOT fbFileRingBuffer.bError THEN
			
			fbFileRingBuffer.A_GetHead(pReadBuff := ADR(arrDataFromFile), cbReadLen := SIZEOF(arrDataFromFile));
			
			iStep:=300;
		END_IF
	300://wait done / take data from array
		IF NOT fbFileRingBuffer.bBusy AND NOT fbFileRingBuffer.bError THEN
			
			M_ST_AlarmHistory_Extract(Input:=arrDataFromFile[AnalizeIndex],Output=>DataToDB);
			//DataToDB:=arrDataFromFile[AnalizeIndex];
			
			//1217//get count of data
			lrTemp:=SIZEOF(ST_AlarmInfo_DB_save);
			udiDataCount:=LREAL_TO_UDINT(fbFileRingBuffer.cbReturn / SIZEOF(ST_AlarmInfo_DB_save));
			
			iStep:=310;
		ELSIF NOT fbFileRingBuffer.bBusy AND fbFileRingBuffer.bError THEN//Empty
			iStep:=600;
		END_IF
	310:// write to DB
	
		IF fbDataUpload_Leo.M_AlarmHistory_Upload(stAlarmInfo:=DataToDB,bExecute:=TRUE) THEN 
		//IF fbAlarmHistory_DB.M_Upload(stAlarmInfo:=DataToDB) THEN
			iStep:=320;
		END_IF
		
	320://wait done
	
		IF NOT fbDataUpload_Leo.AlarmHistoryUpload_Err AND fbDataUpload_Leo.AlarmHistoryUpload_Done THEN
		//IF NOT fbAlarmHistory_DB.bError THEN//write OK
		
			AnalizeIndex:=AnalizeIndex+1;
			
			iStep:=330;
			
		END_IF
		
	330://Check if all data in array Analized
		
		//1217
		//IF AnalizeIndex < GVL.arrArrayLength[eStrIndex]-1 THEN//not done
		IF AnalizeIndex < udiDataCount THEN//not done
			iStep:=300;//go back
		ELSE//array data done
			iStep:=400;//complete this array
		END_IF
		
	400://wait done / remove Head
	
		//1217
		//fbFileRingBuffer.A_RemoveHead(pReadBuff := ADR(arrDataFromFile), cbReadLen := SIZEOF(arrDataFromFile));
		fbFileRingBuffer.A_RemoveHead(pReadBuff := ADR(arrDataFromFile), cbReadLen := fbFileRingBuffer.cbReturn);
		
		iStep:=500;
		
	500://wait done / check if all data got?
		IF NOT fbFileRingBuffer.bBusy AND NOT fbFileRingBuffer.bError THEN
			IF stHeader.nCount > 0 THEN
				iStep:=100;//Go Back
			ELSE
				iStep:=600;//finish
			END_IF
		END_IF
	600://reset file
	
		fbFileRingBuffer.A_Reset();
		
		iStep:=700;
		
	700://wait done / close file
		IF NOT fbFileRingBuffer.bBusy AND NOT fbFileRingBuffer.bError THEN
			
			fbFileRingBuffer.A_Close();
			
			iStep:=800;
		END_IF
	800://wait done
		IF NOT fbFileRingBuffer.bBusy AND NOT fbFileRingBuffer.bError THEN
			
			NovRamData.arrFileRingBuffer_Status[eStrIndex].bFileFull[udiNovRam_BufferIndex][udiFile_Index]:=FALSE;
			
			iStep:=0;
			
		END_IF
		
	
END_CASE
END_METHOD

METHOD M_GetFileName : STRING(255)
VAR_INPUT
	structureType:DINT;
	udiNovRam_BufferIndex:UDINT;
	udiFile_Index:UDINT;
END_VAR
VAR
	tempString:STRING(255);
	tempString2:STRING(255);
	tempFileNo:UDINT;
END_VAR
IF structureType=E_DB_StructureType.AlarmHistory THEN
	tempString:=CONCAT(gvl.arrfileFolder[structureType],'AlarmHistory');
ELSIF structureType=E_DB_StructureType.ProductionHistory THEN
	tempString:=CONCAT(gvl.arrfileFolder[structureType],'ProductionHistory');
ELSIF structureType=E_DB_StructureType.ProductionReport THEN
	tempString:=CONCAT(gvl.arrfileFolder[structureType],'ProductionReport');
ELSIF structureType=E_DB_StructureType.ProductionSummary THEN
	tempString:=CONCAT(gvl.arrfileFolder[structureType],'ProductionSummary');
ELSIF structureType=E_DB_StructureType.SoDuration THEN
	tempString:=CONCAT(gvl.arrfileFolder[structureType],'SoDuration');
ELSIF structureType=E_DB_StructureType.StopCount THEN
	tempString:=CONCAT(gvl.arrfileFolder[structureType],'StopCount');
ELSIF structureType=E_DB_StructureType.RegularCheckResults THEN
	tempString:=CONCAT(gvl.arrfileFolder[structureType],'RegularCheckResults');
END_IF

tempFileNo:=(udiNovRam_BufferIndex) * GVL.FileRingBufferRatio + (udiFile_Index + 1);
tempString2:=CONCAT(tempString,UDINT_TO_STRING(tempFileNo));
M_GetFileName:=CONCAT(tempString2,'.dat');
END_METHOD

{warning 'add method implementation '}
METHOD M_ProductionHistory : BOOL
VAR_INPUT
	
	//udiFileNo:UDINT;
	udiNovRam_BufferIndex:UDINT;
	udiFile_Index:UDINT;
END_VAR
VAR_INST
	arrDataFromFile:ARRAY[0..GVL.arrArrayLength[E_DB_StructureType.ProductionHistory]-1] OF ST_PHI_GroupData_DB;//small
	DataToDB:ST_PHI_GroupData_DB;//large
	AnalizeIndex:UDINT;//should be kept by NovRam
	iStep:INT;
	i:UDINT;
	fbFileRingBuffer: FB_FileRingBuffer := ( sNetId     := '',
                                             sPathName  := '',
                                             ePath      := PATH_GENERIC,
                                             nID        := 1,
                                             cbBuffer   := gvl.arrFileRingBufferSize[E_DB_StructureType.ProductionHistory], //5MB(5*10^6Bytes)
                                             bOverwrite := FALSE,
                                             pWriteBuff := 0,
                                             cbWriteLen := 0,
                                             pReadBuff  := 0,
                                             cbReadLen  := 0,
                                             tTimeout   := T#1S );
	bBusy:BOOL;
	bError:BOOL;
	nErrID:UDINT;
	stHeader:ST_FileRBufferHead;
    //loadData  : ARRAY[0..511] OF BYTE :=[512(0)];
    //cbLoad    : UDINT;
	
	fileName: STRING(255);
	eStrIndex:DINT;
	
	//DB
	fbProductionHistoryInspection_DB		: FB_ProductionHistoryInspection_DB;
	PHI_GroupData_DB : ST_PHI_GroupData_DB;
END_VAR
//Config
eStrIndex:=E_DB_StructureType.ProductionHistory;

fbFileRingBuffer(sPathName:=fileName
				,bBusy=>bBusy,bError=>bError,nErrID=>nErrID
				,stHeader=>stHeader);
				
//DB_Test
fbProductionHistoryInspection_DB(udiDBID:=1);

CASE iStep OF
	0://check if file full 
		IF NovRamData.arrFileRingBuffer_Status[eStrIndex].bFileFull[udiNovRam_BufferIndex][udiFile_Index] = TRUE//file full = should work 
		THEN
			
			fileName:=M_GetFileName(structureType:=eStrIndex
									,udiNovRam_BufferIndex:=udiNovRam_BufferIndex
									,udiFile_Index:=udiFile_Index);
			
			iStep:=100;
		END_IF
	100:// Open file
		
		AnalizeIndex:=0;
		fbFileRingBuffer.A_Open();
		
		iStep:=200;
	200://wait done / read head
		IF NOT fbFileRingBuffer.bBusy AND NOT fbFileRingBuffer.bError THEN
			
			fbFileRingBuffer.A_GetHead(pReadBuff := ADR(arrDataFromFile), cbReadLen := SIZEOF(arrDataFromFile));
			
			iStep:=300;
		END_IF
	300://wait done / take data from array
		IF NOT fbFileRingBuffer.bBusy AND NOT fbFileRingBuffer.bError THEN
			
			M_ST_ProductionHistory_Extract(Input:=arrDataFromFile[AnalizeIndex],Output=>DataToDB);
			//DataToDB:=arrDataFromFile[AnalizeIndex];
			
			iStep:=310;
		ELSIF NOT fbFileRingBuffer.bBusy AND fbFileRingBuffer.bError THEN//Empty
			iStep:=600;
		END_IF
	310:// write to DB
	
		IF fbProductionHistoryInspection_DB.M_Upload(stPHI:=DataToDB) THEN
			iStep:=320;
		END_IF
		
	320://wait done
		
		IF NOT fbProductionHistoryInspection_DB.bError THEN//write OK
		
			AnalizeIndex:=AnalizeIndex+1;
			
			iStep:=330;
			
		ELSE//write failed need to write to log
			;
		END_IF
		
	330://Check if all data in array Analized
		IF AnalizeIndex < GVL.arrArrayLength[eStrIndex]-1 THEN//not done
			iStep:=300;//go back
		ELSE//array data done
			iStep:=400;//complete this array
		END_IF
		
	400://wait done / remove Head
	
		fbFileRingBuffer.A_RemoveHead(pReadBuff := ADR(arrDataFromFile), cbReadLen := SIZEOF(arrDataFromFile));
		
		iStep:=500;
		
	500://wait done / check if all data got?
		IF NOT fbFileRingBuffer.bBusy AND NOT fbFileRingBuffer.bError THEN
			IF stHeader.nCount > 0 THEN
				iStep:=100;//Go Back
			ELSE
				iStep:=600;//finish
			END_IF
		END_IF
	600://reset file
	
		fbFileRingBuffer.A_Reset();
		
		iStep:=700;
		
	700://wait done / close file
		IF NOT fbFileRingBuffer.bBusy AND NOT fbFileRingBuffer.bError THEN
			
			fbFileRingBuffer.A_Close();
			
			iStep:=800;
		END_IF
	800://wait done
		IF NOT fbFileRingBuffer.bBusy AND NOT fbFileRingBuffer.bError THEN
			
			NovRamData.arrFileRingBuffer_Status[eStrIndex].bFileFull[udiNovRam_BufferIndex][udiFile_Index]:=FALSE;
			
			iStep:=0;
			
		END_IF
		
	
END_CASE
END_METHOD

METHOD M_ProductionReport : BOOL
VAR_INPUT
	
	//udiFileNo:UDINT;
	udiNovRam_BufferIndex:UDINT;
	udiFile_Index:UDINT;
END_VAR
VAR_INST
	arrDataFromFile:ARRAY[0..GVL.arrArrayLength[E_DB_StructureType.ProductionReport]-1] OF ST_OEE_ProductionReport;//small
	DataToDB:ST_OEE_ProductionReport;//large
	AnalizeIndex:UDINT;//should be kept by NovRam
	iStep:INT;
	i:UDINT;
	fbFileRingBuffer: FB_FileRingBuffer := ( sNetId     := '',
                                             sPathName  := '',
                                             ePath      := PATH_GENERIC,
                                             nID        := 1,
                                             cbBuffer   := gvl.arrFileRingBufferSize[E_DB_StructureType.ProductionReport], //5MB(5*10^6Bytes)
                                             bOverwrite := FALSE,
                                             pWriteBuff := 0,
                                             cbWriteLen := 0,
                                             pReadBuff  := 0,
                                             cbReadLen  := 0,
                                             tTimeout   := T#1S );
	bBusy:BOOL;
	bError:BOOL;
	nErrID:UDINT;
	stHeader:ST_FileRBufferHead;
    //loadData  : ARRAY[0..511] OF BYTE :=[512(0)];
    //cbLoad    : UDINT;
	
	fileName: STRING(255);
	eStrIndex:DINT;
	fbOEE_ProductionReport_DB:FB_OEE_ProductionReport_DB;
END_VAR
//Config
eStrIndex:=E_DB_StructureType.ProductionReport;

fbFileRingBuffer(sPathName:=fileName
				,bBusy=>bBusy,bError=>bError,nErrID=>nErrID
				,stHeader=>stHeader);
				
CASE iStep OF
	0://check if file full 
		IF NovRamData.arrFileRingBuffer_Status[eStrIndex].bFileFull[udiNovRam_BufferIndex][udiFile_Index] = TRUE//file full = should work 
		THEN
			
			fileName:=M_GetFileName(structureType:=eStrIndex
									,udiNovRam_BufferIndex:=udiNovRam_BufferIndex
									,udiFile_Index:=udiFile_Index);
			
			iStep:=100;
		END_IF
	100:// Open file
		
		AnalizeIndex:=0;
		fbFileRingBuffer.A_Open();
		
		iStep:=200;
	200://wait done / read head
		IF NOT fbFileRingBuffer.bBusy AND NOT fbFileRingBuffer.bError THEN
			
			fbFileRingBuffer.A_GetHead(pReadBuff := ADR(arrDataFromFile), cbReadLen := SIZEOF(arrDataFromFile));
			
			iStep:=300;
		END_IF
	300://wait done / take data from array
		IF NOT fbFileRingBuffer.bBusy AND NOT fbFileRingBuffer.bError THEN
			
			M_ST_ProductionReport_Extract(Input:=arrDataFromFile[AnalizeIndex],Output=>DataToDB);
			//DataToDB:=arrDataFromFile[AnalizeIndex];
			
			iStep:=310;
		ELSIF NOT fbFileRingBuffer.bBusy AND fbFileRingBuffer.bError THEN//Empty
			iStep:=600;
		END_IF
	310:// write to DB
		
		IF fbOEE_ProductionReport_DB.M_Upload(stOeeProductionReport:=DataToDB) THEN
			iStep:=320;
		END_IF
		
	320://wait done
		
		IF NOT fbOEE_ProductionReport_DB.bError THEN//write OK
		
			AnalizeIndex:=AnalizeIndex+1;
			
			iStep:=330;
			
		ELSE//write failed need to write to log
			;
		END_IF
		
		
	330://Check if all data in array Analized
		IF AnalizeIndex < GVL.arrArrayLength[eStrIndex]-1 THEN//not done
			iStep:=300;//go back
		ELSE//array data done
			iStep:=400;//complete this array
		END_IF
		
	400://wait done / remove Head
	
		fbFileRingBuffer.A_RemoveHead(pReadBuff := ADR(arrDataFromFile), cbReadLen := SIZEOF(arrDataFromFile));
		
		iStep:=500;
		
	500://wait done / check if all data got?
		IF NOT fbFileRingBuffer.bBusy AND NOT fbFileRingBuffer.bError THEN
			IF stHeader.nCount > 0 THEN
				iStep:=100;//Go Back
			ELSE
				iStep:=600;//finish
			END_IF
		END_IF
	600://reset file
	
		fbFileRingBuffer.A_Reset();
		
		iStep:=700;
		
	700://wait done / close file
		IF NOT fbFileRingBuffer.bBusy AND NOT fbFileRingBuffer.bError THEN
			
			fbFileRingBuffer.A_Close();
			
			iStep:=800;
		END_IF
	800://wait done
		IF NOT fbFileRingBuffer.bBusy AND NOT fbFileRingBuffer.bError THEN
			
			NovRamData.arrFileRingBuffer_Status[eStrIndex].bFileFull[udiNovRam_BufferIndex][udiFile_Index]:=FALSE;
			
			iStep:=0;
			
		END_IF
		
	
END_CASE
END_METHOD

METHOD M_ProductionSummary : BOOL
VAR_INPUT
	
	//udiFileNo:UDINT;
	udiNovRam_BufferIndex:UDINT;
	udiFile_Index:UDINT;
END_VAR
VAR_INST
	arrDataFromFile:ARRAY[0..GVL.arrArrayLength[E_DB_StructureType.ProductionSummary]-1] OF ST_OEE_ProductionSummary;//small
	DataToDB:ST_OEE_ProductionSummary;//large
	AnalizeIndex:UDINT;//should be kept by NovRam
	iStep:INT;
	i:UDINT;
	fbFileRingBuffer: FB_FileRingBuffer := ( sNetId     := '',
                                             sPathName  := '',
                                             ePath      := PATH_GENERIC,
                                             nID        := 1,
                                             cbBuffer   := gvl.arrFileRingBufferSize[E_DB_StructureType.ProductionSummary], //5MB(5*10^6Bytes)
                                             bOverwrite := FALSE,
                                             pWriteBuff := 0,
                                             cbWriteLen := 0,
                                             pReadBuff  := 0,
                                             cbReadLen  := 0,
                                             tTimeout   := T#1S );
	bBusy:BOOL;
	bError:BOOL;
	nErrID:UDINT;
	stHeader:ST_FileRBufferHead;
    //loadData  : ARRAY[0..511] OF BYTE :=[512(0)];
    //cbLoad    : UDINT;
	
	fileName: STRING(255);
	eStrIndex:DINT;
	fbOEE_ProductionSummary_DB:FB_OEE_ProductionSummary_DB;
END_VAR
//Config
eStrIndex:=E_DB_StructureType.ProductionSummary;

fbFileRingBuffer(sPathName:=fileName
				,bBusy=>bBusy,bError=>bError,nErrID=>nErrID
				,stHeader=>stHeader);
				
CASE iStep OF
	0://check if file full 
		IF NovRamData.arrFileRingBuffer_Status[eStrIndex].bFileFull[udiNovRam_BufferIndex][udiFile_Index] = TRUE//file full = should work 
		THEN
			
			fileName:=M_GetFileName(structureType:=eStrIndex
									,udiNovRam_BufferIndex:=udiNovRam_BufferIndex
									,udiFile_Index:=udiFile_Index);
			
			iStep:=100;
		END_IF
	100:// Open file
		
		AnalizeIndex:=0;
		fbFileRingBuffer.A_Open();
		
		iStep:=200;
	200://wait done / read head
		IF NOT fbFileRingBuffer.bBusy AND NOT fbFileRingBuffer.bError THEN
			
			fbFileRingBuffer.A_GetHead(pReadBuff := ADR(arrDataFromFile), cbReadLen := SIZEOF(arrDataFromFile));
			
			iStep:=300;
		END_IF
	300://wait done / take data from array
		IF NOT fbFileRingBuffer.bBusy AND NOT fbFileRingBuffer.bError THEN
			
			M_ST_ProductionSummary_Extract(Input:=arrDataFromFile[AnalizeIndex],Output=>DataToDB);
			//DataToDB:=arrDataFromFile[AnalizeIndex];
			
			iStep:=310;
		ELSIF NOT fbFileRingBuffer.bBusy AND fbFileRingBuffer.bError THEN//Empty
			iStep:=600;
		END_IF
	310:// write to DB
	
		IF fbOEE_ProductionSummary_DB.M_Upload(stOEEProductionSummary:=DataToDB) THEN
			iStep:=320;
		END_IF
		
	320://wait done
		
			IF NOT fbOEE_ProductionSummary_DB.bError THEN//write OK
			
				AnalizeIndex:=AnalizeIndex+1;
				
				iStep:=330;
				
			ELSE//write failed need to write to log
				;
			END_IF
		
		
	330://Check if all data in array Analized
		IF AnalizeIndex < GVL.arrArrayLength[eStrIndex]-1 THEN//not done
			iStep:=300;//go back
		ELSE//array data done
			iStep:=400;//complete this array
		END_IF
		
	400://wait done / remove Head
	
		fbFileRingBuffer.A_RemoveHead(pReadBuff := ADR(arrDataFromFile), cbReadLen := SIZEOF(arrDataFromFile));
		
		iStep:=500;
		
	500://wait done / check if all data got?
		IF NOT fbFileRingBuffer.bBusy AND NOT fbFileRingBuffer.bError THEN
			IF stHeader.nCount > 0 THEN
				iStep:=100;//Go Back
			ELSE
				iStep:=600;//finish
			END_IF
		END_IF
	600://reset file
	
		fbFileRingBuffer.A_Reset();
		
		iStep:=700;
		
	700://wait done / close file
		IF NOT fbFileRingBuffer.bBusy AND NOT fbFileRingBuffer.bError THEN
			
			fbFileRingBuffer.A_Close();
			
			iStep:=800;
		END_IF
	800://wait done
		IF NOT fbFileRingBuffer.bBusy AND NOT fbFileRingBuffer.bError THEN
			
			NovRamData.arrFileRingBuffer_Status[eStrIndex].bFileFull[udiNovRam_BufferIndex][udiFile_Index]:=FALSE;
			
			iStep:=0;
			
		END_IF
		
	
END_CASE
END_METHOD

METHOD M_RegularCheckResults : BOOL
VAR_INPUT
	
	//udiFileNo:UDINT;
	udiNovRam_BufferIndex:UDINT;
	udiFile_Index:UDINT;
END_VAR
VAR_INST
	arrDataFromFile:ARRAY[0..GVL.arrArrayLength[E_DB_StructureType.RegularCheckResults]-1] OF ST_RegularCheck_Results;//small
	DataToDB:ST_RegularCheck_Results;//large
	AnalizeIndex:UDINT;//should be kept by NovRam
	iStep:INT;
	i:UDINT;
	fbFileRingBuffer: FB_FileRingBuffer := ( sNetId     := '',
                                             sPathName  := '',
                                             ePath      := PATH_GENERIC,
                                             nID        := 1,
                                             cbBuffer   := gvl.arrFileRingBufferSize[E_DB_StructureType.RegularCheckResults], //5MB(5*10^6Bytes)
                                             bOverwrite := FALSE,
                                             pWriteBuff := 0,
                                             cbWriteLen := 0,
                                             pReadBuff  := 0,
                                             cbReadLen  := 0,
                                             tTimeout   := T#1S );
	bBusy:BOOL;
	bError:BOOL;
	nErrID:UDINT;
	stHeader:ST_FileRBufferHead;
    //loadData  : ARRAY[0..511] OF BYTE :=[512(0)];
    //cbLoad    : UDINT;
	
	fileName: STRING(255);
	eStrIndex:DINT;
	fbRegular_Check_Results_DB:FB_Regular_Check_Results_DB;
END_VAR
//Config
eStrIndex:=E_DB_StructureType.RegularCheckResults;

fbFileRingBuffer(sPathName:=fileName
				,bBusy=>bBusy,bError=>bError,nErrID=>nErrID
				,stHeader=>stHeader);
				
CASE iStep OF
	0://check if file full 
		IF NovRamData.arrFileRingBuffer_Status[eStrIndex].bFileFull[udiNovRam_BufferIndex][udiFile_Index] = TRUE//file full = should work 
		THEN
			
			fileName:=M_GetFileName(structureType:=eStrIndex
									,udiNovRam_BufferIndex:=udiNovRam_BufferIndex
									,udiFile_Index:=udiFile_Index);
			
			iStep:=100;
		END_IF
	100:// Open file
		
		AnalizeIndex:=0;
		fbFileRingBuffer.A_Open();
		
		iStep:=200;
	200://wait done / read head
		IF NOT fbFileRingBuffer.bBusy AND NOT fbFileRingBuffer.bError THEN
			
			fbFileRingBuffer.A_GetHead(pReadBuff := ADR(arrDataFromFile), cbReadLen := SIZEOF(arrDataFromFile));
			
			iStep:=300;
		END_IF
	300://wait done / take data from array
		IF NOT fbFileRingBuffer.bBusy AND NOT fbFileRingBuffer.bError THEN
			
			M_ST_RegularCheckResults_Extract(Input:=arrDataFromFile[AnalizeIndex],Output=>DataToDB);
			//DataToDB:=arrDataFromFile[AnalizeIndex];
								
			iStep:=310;
		ELSIF NOT fbFileRingBuffer.bBusy AND fbFileRingBuffer.bError THEN//Empty
			iStep:=600;
		END_IF
	310:// write to DB
		
		IF fbRegular_Check_Results_DB.M_Upload(stRcResults:=DataToDB) THEN
			iStep:=320;
		END_IF
		
	320://wait done
		
		IF NOT fbRegular_Check_Results_DB.bError THEN//write OK
		
			AnalizeIndex:=AnalizeIndex+1;
			
			iStep:=330;
			
		ELSE//write failed need to write to log
			;
		END_IF
		
	330://Check if all data in array Analized
		IF AnalizeIndex < GVL.arrArrayLength[eStrIndex]-1 THEN//not done
			iStep:=300;//go back
		ELSE//array data done
			iStep:=400;//complete this array
		END_IF
		
	400://wait done / remove Head
	
		fbFileRingBuffer.A_RemoveHead(pReadBuff := ADR(arrDataFromFile), cbReadLen := SIZEOF(arrDataFromFile));
		
		iStep:=500;
		
	500://wait done / check if all data got?
		IF NOT fbFileRingBuffer.bBusy AND NOT fbFileRingBuffer.bError THEN
			IF stHeader.nCount > 0 THEN
				iStep:=100;//Go Back
			ELSE
				iStep:=600;//finish
			END_IF
		END_IF
	600://reset file
	
		fbFileRingBuffer.A_Reset();
		
		iStep:=700;
		
	700://wait done / close file
		IF NOT fbFileRingBuffer.bBusy AND NOT fbFileRingBuffer.bError THEN
			
			fbFileRingBuffer.A_Close();
			
			iStep:=800;
		END_IF
	800://wait done
		IF NOT fbFileRingBuffer.bBusy AND NOT fbFileRingBuffer.bError THEN
			
			NovRamData.arrFileRingBuffer_Status[eStrIndex].bFileFull[udiNovRam_BufferIndex][udiFile_Index]:=FALSE;
			
			iStep:=0;
			
		END_IF
		
	
END_CASE
END_METHOD

METHOD M_SoDuration : BOOL
VAR_INPUT
	
